LIN {X 0,Y 397.224,Z 668.821,A -85,B 0,C 180,E1 -11416.703,E2 -11416.703} C_VEL
LIN {X 0,Y 397.214,Z 668.819,A -85,B 0,C 180,E1 -11419.809,E2 -11419.809} C_VEL
LIN {X 0,Y 397.36,Z 668.8,A -85,B 0,C 180,E1 -11422.888,E2 -11422.888} C_VEL
LIN {X 0,Y 397.212,Z 669.008,A -85,B 0,C 180,E1 -11425.433,E2 -11425.433} C_VEL
LIN {X 0,Y 397.512,Z 669.23,A -85,B 0,C 180,E1 -11427.974,E2 -11427.974} C_VEL
LIN {X 0,Y 397.665,Z 669.27,A -85,B 0,C 180,E1 -11430,E2 -11430} C_VEL
LIN {X 0,Y 397.41,Z 669.17,A -85,B 0,C 180,E1 -11433.041,E2 -11433.041} C_VEL
LIN {X 0,Y 397.36,Z 668.8,A -85,B 0,C 180,E1 -11437.112,E2 -11437.112} C_VEL
LIN {X 0,Y 397.214,Z 668.819,A -85,B 0,C 180,E1 -11440.191,E2 -11440.191} C_VEL
LIN {X 0,Y 397.222,Z 668.821,A -85,B 0,C 180,E1 -11443.321,E2 -11443.321} C_VEL
LIN {X 0,Y 397.177,Z 668.825,A -85,B 0,C 180,E1 -11447.155,E2 -11447.155} C_VEL
LIN {X 0,Y 397.098,Z 668.833,A -85,B 0,C 180,E1 -11450.73,E2 -11450.73} C_VEL
LIN {X 0,Y 397.128,Z 668.833,A -85,B 0,C 180,E1 -11454.018,E2 -11454.018} C_VEL
LIN {X 0,Y 397.129,Z 668.83,A -85,B 0,C 180,E1 -11456.329,E2 -11456.329} C_VEL
LIN {X 0,Y 396.46,Z 668.913,A -85,B 0,C 180,E1 -11457.176,E2 -11457.176} C_VEL
LIN {X 0,Y 393.587,Z 669.271,A -85,B 0,C 180,E1 -11458.552,E2 -11458.552} C_VEL
LIN {X 0,Y 391.15,Z 669.576,A -85,B 0,C 180,E1 -11459.663,E2 -11459.663} C_VEL
LIN {X 0,Y 390.098,Z 669.707,A -85,B 0,C 180,E1 -11460.523,E2 -11460.523} C_VEL
LIN {X 0,Y 390.01,Z 669.714,A -85,B 0,C 180,E1 -11460.814,E2 -11460.814} C_VEL
LIN {X 0,Y 390.062,Z 669.71,A -85,B 0,C 180,E1 -11464.024,E2 -11464.024} C_VEL
LIN {X 0,Y 390.04,Z 669.713,A -85,B 0,C 180,E1 -11467.551,E2 -11467.551} C_VEL
LIN {X 0,Y 390.07,Z 669.71,A -85,B 0,C 180,E1 -11470.824,E2 -11470.824} C_VEL
LIN {X 0,Y 390.052,Z 669.711,A -85,B 0,C 180,E1 -11473.886,E2 -11473.886} C_VEL
LIN {X 0,Y 390.108,Z 669.706,A -85,B 0,C 180,E1 -11476.797,E2 -11476.797} C_VEL
LIN {X 0,Y 390.07,Z 669.71,A -85,B 0,C 180,E1 -11479.563,E2 -11479.563} C_VEL
LIN {X 0,Y 390.039,Z 669.686,A -85,B 0,C 180,E1 -11482.448,E2 -11482.448} C_VEL
LIN {X 0,Y 390.059,Z 669.698,A -85,B 0,C 180,E1 -11485.975,E2 -11485.975} C_VEL
LIN {X 0,Y 390.042,Z 669.68,A -85,B 0,C 180,E1 -11489.868,E2 -11489.868} C_VEL
LIN {X 0,Y 390.104,Z 669.682,A -85,B 0,C 180,E1 -11493.232,E2 -11493.232} C_VEL
LIN {X 0,Y 390.102,Z 669.699,A -85,B 0,C 180,E1 -11496.748,E2 -11496.748} C_VEL
LIN {X 0,Y 390.121,Z 669.704,A -85,B 0,C 180,E1 -11499.984,E2 -11499.984} C_VEL
LIN {X 0,Y 390.128,Z 669.69,A -85,B 0,C 180,E1 -11503.248,E2 -11503.248} C_VEL
LIN {X 0,Y 390.185,Z 669.677,A -85,B 0,C 180,E1 -11506.562,E2 -11506.562} C_VEL
LIN {X 0,Y 390.199,Z 669.684,A -85,B 0,C 180,E1 -11510.671,E2 -11510.671} C_VEL
LIN {X 0,Y 390.328,Z 669.669,A -85,B 0,C 180,E1 -11513.798,E2 -11513.798} C_VEL
LIN {X 0,Y 390.411,Z 669.649,A -85,B 0,C 180,E1 -11517.937,E2 -11517.937} C_VEL
LIN {X 0,Y 390.542,Z 669.648,A -85,B 0,C 180,E1 -11520,E2 -11520} C_VEL
LIN {X 0,Y 390.308,Z 669.665,A -85,B 0,C 180,E1 -11523.097,E2 -11523.097} C_VEL
LIN {X 0,Y 390.33,Z 669.673,A -85,B 0,C 180,E1 -11526.202,E2 -11526.202} C_VEL
LIN {X 0,Y 390.201,Z 669.685,A -85,B 0,C 180,E1 -11529.329,E2 -11529.329} C_VEL
LIN {X 0,Y 390.17,Z 669.682,A -85,B 0,C 180,E1 -11532.483,E2 -11532.483} C_VEL
LIN {X 0,Y 390.131,Z 669.698,A -85,B 0,C 180,E1 -11535.677,E2 -11535.677} C_VEL
LIN {X 0,Y 390.108,Z 669.695,A -85,B 0,C 180,E1 -11538.922,E2 -11538.922} C_VEL
LIN {X 0,Y 390.032,Z 669.699,A -85,B 0,C 180,E1 -11542.235,E2 -11542.235} C_VEL
LIN {X 0,Y 390.111,Z 669.696,A -85,B 0,C 180,E1 -11545.744,E2 -11545.744} C_VEL
LIN {X 0,Y 390.056,Z 669.66,A -85,B 0,C 180,E1 -11549.11,E2 -11549.11} C_VEL
LIN {X 0,Y 390.037,Z 669.712,A -85,B 0,C 180,E1 -11552.722,E2 -11552.722} C_VEL
LIN {X 0,Y 390.051,Z 669.68,A -85,B 0,C 180,E1 -11555.826,E2 -11555.826} C_VEL
LIN {X 0,Y 390.069,Z 669.707,A -85,B 0,C 180,E1 -11559.22,E2 -11559.22} C_VEL
LIN {X 0,Y 390.117,Z 669.688,A -85,B 0,C 180,E1 -11562.388,E2 -11562.388} C_VEL
LIN {X 0,Y 390.059,Z 669.69,A -85,B 0,C 180,E1 -11565.358,E2 -11565.358} C_VEL
LIN {X 0,Y 390.068,Z 669.864,A -85,B 0,C 180,E1 -11569.083,E2 -11569.083} C_VEL
LIN {X 0,Y 393.041,Z 680.441,A -85,B 0,C 180,E1 -11571.884,E2 -11571.884} C_VEL
LIN {X 0,Y 395.697,Z 690.609,A -85,B 0,C 180,E1 -11574.336,E2 -11574.336} C_VEL
LIN {X 0,Y 404.177,Z 707.9,A -85,B 0,C 180,E1 -11575.584,E2 -11575.584} C_VEL
LIN {X 0,Y 406.863,Z 714.125,A -85,B 0,C 180,E1 -11575.97,E2 -11575.97} C_VEL
LIN {X 0,Y 412.259,Z 737.158,A -85,B 0,C 180,E1 -11576.941,E2 -11576.941} C_VEL
LIN {X 0,Y 409.574,Z 850.002,A -85,B 0,C 180,E1 -11578.982,E2 -11578.982} C_VEL
LIN {X 0,Y 408.459,Z 894.918,A -85,B 0,C 180,E1 -11579.824,E2 -11579.824} C_VEL
LIN {X 0,Y 407.68,Z 907.428,A -85,B 0,C 180,E1 -11580.148,E2 -11580.148} C_VEL
LIN {X 0,Y 406.718,Z 919.552,A -85,B 0,C 180,E1 -11580.569,E2 -11580.569} C_VEL
LIN {X 0,Y 405.755,Z 931.929,A -85,B 0,C 180,E1 -11581.131,E2 -11581.131} C_VEL
LIN {X 0,Y 404.553,Z 943.316,A -85,B 0,C 180,E1 -11581.746,E2 -11581.746} C_VEL
LIN {X 0,Y 402.984,Z 957.059,A -85,B 0,C 180,E1 -11582.657,E2 -11582.657} C_VEL
LIN {X 0,Y 401.59,Z 968.362,A -85,B 0,C 180,E1 -11583.546,E2 -11583.546} C_VEL
LIN {X 0,Y 399.899,Z 980.294,A -85,B 0,C 180,E1 -11584.636,E2 -11584.636} C_VEL
LIN {X 0,Y 398.332,Z 991.097,A -85,B 0,C 180,E1 -11585.782,E2 -11585.782} C_VEL
LIN {X 0,Y 396.667,Z 1002.013,A -85,B 0,C 180,E1 -11587.119,E2 -11587.119} C_VEL
LIN {X 0,Y 395.292,Z 1010.87,A -85,B 0,C 180,E1 -11588.352,E2 -11588.352} C_VEL
LIN {X 0,Y 393.836,Z 1020.607,A -85,B 0,C 180,E1 -11589.909,E2 -11589.909} C_VEL
LIN {X 0,Y 392.506,Z 1029.848,A -85,B 0,C 180,E1 -11591.62,E2 -11591.62} C_VEL
LIN {X 0,Y 391.471,Z 1037.738,A -85,B 0,C 180,E1 -11593.307,E2 -11593.307} C_VEL
LIN {X 0,Y 390.576,Z 1044.167,A -85,B 0,C 180,E1 -11594.876,E2 -11594.876} C_VEL
LIN {X 0,Y 389.798,Z 1051.393,A -85,B 0,C 180,E1 -11596.964,E2 -11596.964} C_VEL
LIN {X 0,Y 389.384,Z 1056.079,A -85,B 0,C 180,E1 -11598.549,E2 -11598.549} C_VEL
LIN {X 0,Y 388.957,Z 1061.172,A -85,B 0,C 180,E1 -11600.641,E2 -11600.641} C_VEL
LIN {X 0,Y 388.806,Z 1065.168,A -85,B 0,C 180,E1 -11602.731,E2 -11602.731} C_VEL
LIN {X 0,Y 388.737,Z 1067.048,A -85,B 0,C 180,E1 -11603.905,E2 -11603.905} C_VEL
LIN {X 0,Y 388.657,Z 1069.301,A -85,B 0,C 180,E1 -11605.852,E2 -11605.852} C_VEL
LIN {X 0,Y 388.649,Z 1070.765,A -85,B 0,C 180,E1 -11607.927,E2 -11607.927} C_VEL
LIN {X 0,Y 388.704,Z 1071.251,A -85,B 0,C 180,E1 -11610,E2 -11610} C_VEL
LIN {X 0,Y 388.649,Z 1070.765,A -85,B 0,C 180,E1 -11612.073,E2 -11612.073} C_VEL
LIN {X 0,Y 388.657,Z 1069.301,A -85,B 0,C 180,E1 -11614.148,E2 -11614.148} C_VEL
LIN {X 0,Y 388.757,Z 1066.839,A -85,B 0,C 180,E1 -11616.227,E2 -11616.227} C_VEL
LIN {X 0,Y 388.897,Z 1062.26,A -85,B 0,C 180,E1 -11618.836,E2 -11618.836} C_VEL
LIN {X 0,Y 389.073,Z 1058.772,A -85,B 0,C 180,E1 -11620.406,E2 -11620.406} C_VEL
LIN {X 0,Y 389.66,Z 1053.051,A -85,B 0,C 180,E1 -11622.499,E2 -11622.499} C_VEL
LIN {X 0,Y 390.151,Z 1047.991,A -85,B 0,C 180,E1 -11624.074,E2 -11624.074} C_VEL
LIN {X 0,Y 391.109,Z 1039.958,A -85,B 0,C 180,E1 -11626.172,E2 -11626.172} C_VEL
LIN {X 0,Y 392.109,Z 1032.976,A -85,B 0,C 180,E1 -11627.74,E2 -11627.74} C_VEL
LIN {X 0,Y 393.19,Z 1025.004,A -85,B 0,C 180,E1 -11629.309,E2 -11629.309} C_VEL
LIN {X 0,Y 394.569,Z 1015.889,A -85,B 0,C 180,E1 -11630.869,E2 -11630.869} C_VEL
LIN {X 0,Y 396.135,Z 1005.854,A -85,B 0,C 180,E1 -11632.359,E2 -11632.359} C_VEL
LIN {X 0,Y 397.641,Z 995.45,A -85,B 0,C 180,E1 -11633.708,E2 -11633.708} C_VEL
LIN {X 0,Y 399.365,Z 984.036,A -85,B 0,C 180,E1 -11634.982,E2 -11634.982} C_VEL
LIN {X 0,Y 400.786,Z 973.609,A -85,B 0,C 180,E1 -11636,E2 -11636} C_VEL
LIN {X 0,Y 402.435,Z 961.583,A -85,B 0,C 180,E1 -11637.003,E2 -11637.003} C_VEL
LIN {X 0,Y 403.884,Z 949.459,A -85,B 0,C 180,E1 -11637.867,E2 -11637.867} C_VEL
LIN {X 0,Y 405.278,Z 936.716,A -85,B 0,C 180,E1 -11638.623,E2 -11638.623} C_VEL
LIN {X 0,Y 406.417,Z 923.283,A -85,B 0,C 180,E1 -11639.278,E2 -11639.278} C_VEL
LIN {X 0,Y 407.461,Z 910.365,A -85,B 0,C 180,E1 -11639.763,E2 -11639.763} C_VEL
LIN {X 0,Y 408.373,Z 896.659,A -85,B 0,C 180,E1 -11640.139,E2 -11640.139} C_VEL
LIN {X 0,Y 409.085,Z 870.937,A -85,B 0,C 180,E1 -11640.64,E2 -11640.64} C_VEL
LIN {X 0,Y 412.265,Z 737.158,A -85,B 0,C 180,E1 -11643.059,E2 -11643.059} C_VEL
LIN {X 0,Y 406.66,Z 713.318,A -85,B 0,C 180,E1 -11644.065,E2 -11644.065} C_VEL
LIN {X 0,Y 397.258,Z 693.815,A -85,B 0,C 180,E1 -11645.402,E2 -11645.402} C_VEL
LIN {X 0,Y 395.726,Z 690.524,A -85,B 0,C 180,E1 -11645.67,E2 -11645.67} C_VEL
LIN {X 0,Y 391.984,Z 676.49,A -85,B 0,C 180,E1 -11649.122,E2 -11649.122} C_VEL
LIN {X 0,Y 390.049,Z 669.745,A -85,B 0,C 180,E1 -11650.968,E2 -11650.968} C_VEL
LIN {X 0,Y 390.059,Z 669.689,A -85,B 0,C 180,E1 -11654.642,E2 -11654.642} C_VEL
LIN {X 0,Y 390.117,Z 669.688,A -85,B 0,C 180,E1 -11657.612,E2 -11657.612} C_VEL
LIN {X 0,Y 390.09,Z 669.705,A -85,B 0,C 180,E1 -11660.908,E2 -11660.908} C_VEL
LIN {X 0,Y 390.079,Z 669.679,A -85,B 0,C 180,E1 -11664.792,E2 -11664.792} C_VEL
LIN {X 0,Y 390.02,Z 669.706,A -85,B 0,C 180,E1 -11668.495,E2 -11668.495} C_VEL
LIN {X 0,Y 390.11,Z 669.657,A -85,B 0,C 180,E1 -11672.069,E2 -11672.069} C_VEL
LIN {X 0,Y 390.072,Z 669.707,A -85,B 0,C 180,E1 -11675.519,E2 -11675.519} C_VEL
LIN {X 0,Y 390.057,Z 669.708,A -85,B 0,C 180,E1 -11678.878,E2 -11678.878} C_VEL
LIN {X 0,Y 390.122,Z 669.689,A -85,B 0,C 180,E1 -11682.166,E2 -11682.166} C_VEL
LIN {X 0,Y 390.138,Z 669.695,A -85,B 0,C 180,E1 -11685.392,E2 -11685.392} C_VEL
LIN {X 0,Y 390.152,Z 669.692,A -85,B 0,C 180,E1 -11688.571,E2 -11688.571} C_VEL
LIN {X 0,Y 390.299,Z 669.66,A -85,B 0,C 180,E1 -11692.03,E2 -11692.03} C_VEL
LIN {X 0,Y 390.225,Z 669.688,A -85,B 0,C 180,E1 -11694.833,E2 -11694.833} C_VEL
LIN {X 0,Y 390.411,Z 669.654,A -85,B 0,C 180,E1 -11697.936,E2 -11697.936} C_VEL
LIN {X 0,Y 390.542,Z 669.647,A -85,B 0,C 180,E1 -11700,E2 -11700} C_VEL
LIN {X 0,Y 390.308,Z 669.662,A -85,B 0,C 180,E1 -11703.096,E2 -11703.096} C_VEL
LIN {X 0,Y 390.3,Z 669.67,A -85,B 0,C 180,E1 -11706.58,E2 -11706.58} C_VEL
LIN {X 0,Y 390.199,Z 669.686,A -85,B 0,C 180,E1 -11709.329,E2 -11709.329} C_VEL
LIN {X 0,Y 390.185,Z 669.678,A -85,B 0,C 180,E1 -11713.438,E2 -11713.438} C_VEL
LIN {X 0,Y 390.139,Z 669.687,A -85,B 0,C 180,E1 -11717.308,E2 -11717.308} C_VEL
LIN {X 0,Y 390.106,Z 669.702,A -85,B 0,C 180,E1 -11720.481,E2 -11720.481} C_VEL
LIN {X 0,Y 390.101,Z 669.699,A -85,B 0,C 180,E1 -11723.35,E2 -11723.35} C_VEL
LIN {X 0,Y 390.104,Z 669.681,A -85,B 0,C 180,E1 -11726.768,E2 -11726.768} C_VEL
LIN {X 0,Y 390.034,Z 669.684,A -85,B 0,C 180,E1 -11730.3,E2 -11730.3} C_VEL
LIN {X 0,Y 390.059,Z 669.698,A -85,B 0,C 180,E1 -11734.025,E2 -11734.025} C_VEL
LIN {X 0,Y 390.039,Z 669.686,A -85,B 0,C 180,E1 -11737.552,E2 -11737.552} C_VEL
LIN {X 0,Y 390.075,Z 669.71,A -85,B 0,C 180,E1 -11740.826,E2 -11740.826} C_VEL
LIN {X 0,Y 390.096,Z 669.706,A -85,B 0,C 180,E1 -11743.894,E2 -11743.894} C_VEL
LIN {X 0,Y 390.073,Z 669.71,A -85,B 0,C 180,E1 -11747.62,E2 -11747.62} C_VEL
LIN {X 0,Y 390.088,Z 669.708,A -85,B 0,C 180,E1 -11750.909,E2 -11750.909} C_VEL
LIN {X 0,Y 390.079,Z 669.708,A -85,B 0,C 180,E1 -11754.794,E2 -11754.794} C_VEL
LIN {X 0,Y 390.021,Z 669.714,A -85,B 0,C 180,E1 -11758.496,E2 -11758.496} C_VEL
LIN {X 0,Y 390.112,Z 669.705,A -85,B 0,C 180,E1 -11762.07,E2 -11762.07} C_VEL
LIN {X 0,Y 390.075,Z 669.708,A -85,B 0,C 180,E1 -11765.52,E2 -11765.52} C_VEL
LIN {X 0,Y 390.051,Z 669.712,A -85,B 0,C 180,E1 -11768.878,E2 -11768.878} C_VEL
LIN {X 0,Y 390.124,Z 669.702,A -85,B 0,C 180,E1 -11772.167,E2 -11772.167} C_VEL
LIN {X 0,Y 390.14,Z 669.731,A -85,B 0,C 180,E1 -11775.393,E2 -11775.393} C_VEL
LIN {X 0,Y 390.278,Z 670.28,A -85,B 0,C 180,E1 -11776.757,E2 -11776.757} C_VEL
LIN {X 0,Y 390.794,Z 671.827,A -85,B 0,C 180,E1 -11777.867,E2 -11777.867} C_VEL
LIN {X 0,Y 392.016,Z 673.68,A -85,B 0,C 180,E1 -11779.411,E2 -11779.411} C_VEL
LIN {X 0,Y 393.321,Z 674.699,A -85,B 0,C 180,E1 -11781.264,E2 -11781.264} C_VEL
LIN {X 0,Y 394.824,Z 675.448,A -85,B 0,C 180,E1 -11783.869,E2 -11783.869} C_VEL
LIN {X 0,Y 395.643,Z 676.056,A -85,B 0,C 180,E1 -11785.926,E2 -11785.926} C_VEL
LIN {X 0,Y 396.111,Z 676.191,A -85,B 0,C 180,E1 -11787.966,E2 -11787.966} C_VEL
LIN {X 0,Y 396.315,Z 676.238,A -85,B 0,C 180,E1 -11790,E2 -11790} C_VEL
LIN {X 0,Y 396.112,Z 676.191,A -85,B 0,C 180,E1 -11792.034,E2 -11792.034} C_VEL
LIN {X 0,Y 395.45,Z 675.884,A -85,B 0,C 180,E1 -11794.587,E2 -11794.587} C_VEL
LIN {X 0,Y 394.284,Z 675.199,A -85,B 0,C 180,E1 -11797.167,E2 -11797.167} C_VEL
LIN {X 0,Y 392.652,Z 674.256,A -85,B 0,C 180,E1 -11799.699,E2 -11799.699} C_VEL
LIN {X 0,Y 391.359,Z 672.872,A -85,B 0,C 180,E1 -11801.393,E2 -11801.393} C_VEL
LIN {X 0,Y 390.326,Z 670.548,A -85,B 0,C 180,E1 -11802.973,E2 -11802.973} C_VEL
LIN {X 0,Y 390.138,Z 669.78,A -85,B 0,C 180,E1 -11804.075,E2 -11804.075} C_VEL
LIN {X 0,Y 390.144,Z 669.702,A -85,B 0,C 180,E1 -11807.307,E2 -11807.307} C_VEL
LIN {X 0,Y 390.082,Z 669.707,A -85,B 0,C 180,E1 -11810.47,E2 -11810.47} C_VEL
LIN {X 0,Y 390.084,Z 669.707,A -85,B 0,C 180,E1 -11813.35,E2 -11813.35} C_VEL
LIN {X 0,Y 390.108,Z 669.706,A -85,B 0,C 180,E1 -11816.768,E2 -11816.768} C_VEL
LIN {X 0,Y 390.038,Z 669.713,A -85,B 0,C 180,E1 -11820.299,E2 -11820.299} C_VEL
LIN {X 0,Y 390.01,Z 669.714,A -85,B 0,C 180,E1 -11820.814,E2 -11820.814} C_VEL
LIN {X 0,Y 389.336,Z 669.8,A -85,B 0,C 180,E1 -11821.676,E2 -11821.676} C_VEL
LIN {X 0,Y 386.486,Z 670.155,A -85,B 0,C 180,E1 -11823.078,E2 -11823.078} C_VEL
LIN {X 0,Y 384.087,Z 670.454,A -85,B 0,C 180,E1 -11824.211,E2 -11824.211} C_VEL
LIN {X 0,Y 383.069,Z 670.582,A -85,B 0,C 180,E1 -11825.087,E2 -11825.087} C_VEL
LIN {X 0,Y 382.993,Z 670.588,A -85,B 0,C 180,E1 -11825.383,E2 -11825.383} C_VEL
LIN {X 0,Y 383.001,Z 670.59,A -85,B 0,C 180,E1 -11828.6,E2 -11828.6} C_VEL
LIN {X 0,Y 383.006,Z 670.589,A -85,B 0,C 180,E1 -11831.343,E2 -11831.343} C_VEL
LIN {X 0,Y 383,Z 670.591,A -85,B 0,C 180,E1 -11834.305,E2 -11834.305} C_VEL
LIN {X 0,Y 383.067,Z 670.583,A -85,B 0,C 180,E1 -11837.249,E2 -11837.249} C_VEL
LIN {X 0,Y 383.014,Z 670.588,A -85,B 0,C 180,E1 -11840.412,E2 -11840.412} C_VEL
LIN {X 0,Y 383.018,Z 670.546,A -85,B 0,C 180,E1 -11844.044,E2 -11844.044} C_VEL
LIN {X 0,Y 382.979,Z 670.593,A -85,B 0,C 180,E1 -11847.577,E2 -11847.577} C_VEL
LIN {X 0,Y 382.987,Z 670.549,A -85,B 0,C 180,E1 -11850.3,E2 -11850.3} C_VEL
LIN {X 0,Y 383.047,Z 670.548,A -85,B 0,C 180,E1 -11852.698,E2 -11852.698} C_VEL
LIN {X 0,Y 383.034,Z 670.581,A -85,B 0,C 180,E1 -11856.193,E2 -11856.193} C_VEL
LIN {X 0,Y 383.072,Z 670.579,A -85,B 0,C 180,E1 -11859.6,E2 -11859.6} C_VEL
LIN {X 0,Y 383.095,Z 670.565,A -85,B 0,C 180,E1 -11862.931,E2 -11862.931} C_VEL
LIN {X 0,Y 383.116,Z 670.558,A -85,B 0,C 180,E1 -11866.464,E2 -11866.464} C_VEL
LIN {X 0,Y 383.145,Z 670.565,A -85,B 0,C 180,E1 -11870.498,E2 -11870.498} C_VEL
LIN {X 0,Y 383.282,Z 670.546,A -85,B 0,C 180,E1 -11873.684,E2 -11873.684} C_VEL
LIN {X 0,Y 383.379,Z 670.524,A -85,B 0,C 180,E1 -11877.899,E2 -11877.899} C_VEL
LIN {X 0,Y 383.511,Z 670.524,A -85,B 0,C 180,E1 -11880,E2 -11880} C_VEL
LIN {X 0,Y 383.244,Z 670.544,A -85,B 0,C 180,E1 -11883.154,E2 -11883.154} C_VEL
LIN {X 0,Y 383.284,Z 670.551,A -85,B 0,C 180,E1 -11886.317,E2 -11886.317} C_VEL
LIN {X 0,Y 383.148,Z 670.566,A -85,B 0,C 180,E1 -11889.502,E2 -11889.502} C_VEL
LIN {X 0,Y 383.133,Z 670.557,A -85,B 0,C 180,E1 -11892.716,E2 -11892.716} C_VEL
LIN {X 0,Y 383.072,Z 670.576,A -85,B 0,C 180,E1 -11895.974,E2 -11895.974} C_VEL
LIN {X 0,Y 383.063,Z 670.576,A -85,B 0,C 180,E1 -11899.284,E2 -11899.284} C_VEL
LIN {X 0,Y 383,Z 670.574,A -85,B 0,C 180,E1 -11902.665,E2 -11902.665} C_VEL
LIN {X 0,Y 383.072,Z 670.569,A -85,B 0,C 180,E1 -11906.124,E2 -11906.124} C_VEL
LIN {X 0,Y 383.042,Z 670.532,A -85,B 0,C 180,E1 -11908.493,E2 -11908.493} C_VEL
LIN {X 0,Y 383.004,Z 670.589,A -85,B 0,C 180,E1 -11912.15,E2 -11912.15} C_VEL
LIN {X 0,Y 383.011,Z 670.565,A -85,B 0,C 180,E1 -11914.669,E2 -11914.669} C_VEL
LIN {X 0,Y 382.998,Z 670.585,A -85,B 0,C 180,E1 -11917.905,E2 -11917.905} C_VEL
LIN {X 0,Y 383.041,Z 670.558,A -85,B 0,C 180,E1 -11921.34,E2 -11921.34} C_VEL
LIN {X 0,Y 383.032,Z 670.575,A -85,B 0,C 180,E1 -11924.31,E2 -11924.31} C_VEL
LIN {X 0,Y 382.983,Z 670.585,A -85,B 0,C 180,E1 -11927.95,E2 -11927.95} C_VEL
LIN {X 0,Y 383.025,Z 670.88,A -85,B 0,C 180,E1 -11928.499,E2 -11928.499} C_VEL
LIN {X 0,Y 386.182,Z 681.98,A -85,B 0,C 180,E1 -11931.494,E2 -11931.494} C_VEL
LIN {X 0,Y 388.446,Z 690.413,A -85,B 0,C 180,E1 -11933.574,E2 -11933.574} C_VEL
LIN {X 0,Y 397.258,Z 708.158,A -85,B 0,C 180,E1 -11934.908,E2 -11934.908} C_VEL
LIN {X 0,Y 401.315,Z 717.115,A -85,B 0,C 180,E1 -11935.502,E2 -11935.502} C_VEL
LIN {X 0,Y 406.335,Z 738.734,A -85,B 0,C 180,E1 -11936.432,E2 -11936.432} C_VEL
LIN {X 0,Y 402.43,Z 891.118,A -85,B 0,C 180,E1 -11939.23,E2 -11939.23} C_VEL
LIN {X 0,Y 401.727,Z 904.285,A -85,B 0,C 180,E1 -11939.55,E2 -11939.55} C_VEL
LIN {X 0,Y 400.613,Z 918.6,A -85,B 0,C 180,E1 -11940.039,E2 -11940.039} C_VEL
LIN {X 0,Y 399.502,Z 931.722,A -85,B 0,C 180,E1 -11940.636,E2 -11940.636} C_VEL
LIN {X 0,Y 398.284,Z 943.109,A -85,B 0,C 180,E1 -11941.26,E2 -11941.26} C_VEL
LIN {X 0,Y 396.71,Z 956.348,A -85,B 0,C 180,E1 -11942.145,E2 -11942.145} C_VEL
LIN {X 0,Y 395.136,Z 968.521,A -85,B 0,C 180,E1 -11943.116,E2 -11943.116} C_VEL
LIN {X 0,Y 393.43,Z 980.087,A -85,B 0,C 180,E1 -11944.189,E2 -11944.189} C_VEL
LIN {X 0,Y 391.774,Z 990.889,A -85,B 0,C 180,E1 -11945.35,E2 -11945.35} C_VEL
LIN {X 0,Y 390.124,Z 1001.391,A -85,B 0,C 180,E1 -11946.652,E2 -11946.652} C_VEL
LIN {X 0,Y 388.608,Z 1010.662,A -85,B 0,C 180,E1 -11947.96,E2 -11947.96} C_VEL
LIN {X 0,Y 387.069,Z 1020.398,A -85,B 0,C 180,E1 -11949.543,E2 -11949.543} C_VEL
LIN {X 0,Y 385.72,Z 1029.432,A -85,B 0,C 180,E1 -11951.24,E2 -11951.24} C_VEL
LIN {X 0,Y 384.597,Z 1037.53,A -85,B 0,C 180,E1 -11953,E2 -11953} C_VEL
LIN {X 0,Y 383.627,Z 1043.959,A -85,B 0,C 180,E1 -11954.596,E2 -11954.596} C_VEL
LIN {X 0,Y 382.827,Z 1050.972,A -85,B 0,C 180,E1 -11956.651,E2 -11956.651} C_VEL
LIN {X 0,Y 382.343,Z 1055.871,A -85,B 0,C 180,E1 -11958.335,E2 -11958.335} C_VEL
LIN {X 0,Y 381.898,Z 1060.965,A -85,B 0,C 180,E1 -11960.467,E2 -11960.467} C_VEL
LIN {X 0,Y 381.708,Z 1064.961,A -85,B 0,C 180,E1 -11962.595,E2 -11962.595} C_VEL
LIN {X 0,Y 381.655,Z 1067.021,A -85,B 0,C 180,E1 -11963.924,E2 -11963.924} C_VEL
LIN {X 0,Y 381.582,Z 1069.095,A -85,B 0,C 180,E1 -11965.775,E2 -11965.775} C_VEL
LIN {X 0,Y 381.547,Z 1070.559,A -85,B 0,C 180,E1 -11967.889,E2 -11967.889} C_VEL
LIN {X 0,Y 381.635,Z 1071.047,A -85,B 0,C 180,E1 -11970,E2 -11970} C_VEL
LIN {X 0,Y 381.547,Z 1070.559,A -85,B 0,C 180,E1 -11972.111,E2 -11972.111} C_VEL
LIN {X 0,Y 381.582,Z 1069.095,A -85,B 0,C 180,E1 -11974.225,E2 -11974.225} C_VEL
LIN {X 0,Y 381.662,Z 1066.633,A -85,B 0,C 180,E1 -11976.343,E2 -11976.343} C_VEL
LIN {X 0,Y 381.821,Z 1062.052,A -85,B 0,C 180,E1 -11979.001,E2 -11979.001} C_VEL
LIN {X 0,Y 382.032,Z 1058.565,A -85,B 0,C 180,E1 -11980.6,E2 -11980.6} C_VEL
LIN {X 0,Y 382.65,Z 1052.843,A -85,B 0,C 180,E1 -11982.732,E2 -11982.732} C_VEL
LIN {X 0,Y 383.169,Z 1047.782,A -85,B 0,C 180,E1 -11984.336,E2 -11984.336} C_VEL
LIN {X 0,Y 384.207,Z 1039.75,A -85,B 0,C 180,E1 -11986.47,E2 -11986.47} C_VEL
LIN {X 0,Y 385.206,Z 1032.766,A -85,B 0,C 180,E1 -11988.068,E2 -11988.068} C_VEL
LIN {X 0,Y 386.381,Z 1024.795,A -85,B 0,C 180,E1 -11989.663,E2 -11989.663} C_VEL
LIN {X 0,Y 387.837,Z 1015.681,A -85,B 0,C 180,E1 -11991.248,E2 -11991.248} C_VEL
LIN {X 0,Y 389.42,Z 1006.053,A -85,B 0,C 180,E1 -11992.706,E2 -11992.706} C_VEL
LIN {X 0,Y 391.093,Z 995.242,A -85,B 0,C 180,E1 -11994.13,E2 -11994.13} C_VEL
LIN {X 0,Y 392.682,Z 985.075,A -85,B 0,C 180,E1 -11995.296,E2 -11995.296} C_VEL
LIN {X 0,Y 394.373,Z 973.402,A -85,B 0,C 180,E1 -11996.456,E2 -11996.456} C_VEL
LIN {X 0,Y 396.067,Z 961.376,A -85,B 0,C 180,E1 -11997.474,E2 -11997.474} C_VEL
LIN {X 0,Y 397.579,Z 949.053,A -85,B 0,C 180,E1 -11998.363,E2 -11998.363} C_VEL
LIN {X 0,Y 399.022,Z 936.509,A -85,B 0,C 180,E1 -11999.114,E2 -11999.114} C_VEL
LIN {X 0,Y 400.223,Z 923.077,A -85,B 0,C 180,E1 -11999.776,E2 -11999.776} C_VEL
LIN {X 0,Y 401.321,Z 910.16,A -85,B 0,C 180,E1 -12000.266,E2 -12000.266} C_VEL
LIN {X 0,Y 402.237,Z 896.826,A -85,B 0,C 180,E1 -12000.638,E2 -12000.638} C_VEL
LIN {X 0,Y 402.977,Z 871.625,A -85,B 0,C 180,E1 -12001.138,E2 -12001.138} C_VEL
LIN {X 0,Y 406.361,Z 738.759,A -85,B 0,C 180,E1 -12003.565,E2 -12003.565} C_VEL
LIN {X 0,Y 401.03,Z 716.167,A -85,B 0,C 180,E1 -12004.546,E2 -12004.546} C_VEL
LIN {X 0,Y 392.191,Z 697.813,A -85,B 0,C 180,E1 -12005.837,E2 -12005.837} C_VEL
LIN {X 0,Y 388.368,Z 690.209,A -85,B 0,C 180,E1 -12006.456,E2 -12006.456} C_VEL
LIN {X 0,Y 385.491,Z 679.253,A -85,B 0,C 180,E1 -12009.211,E2 -12009.211} C_VEL
LIN {X 0,Y 383.019,Z 670.855,A -85,B 0,C 180,E1 -12011.5,E2 -12011.5} C_VEL
LIN {X 0,Y 382.983,Z 670.585,A -85,B 0,C 180,E1 -12012.05,E2 -12012.05} C_VEL
LIN {X 0,Y 383.036,Z 670.576,A -85,B 0,C 180,E1 -12015.795,E2 -12015.795} C_VEL
LIN {X 0,Y 383.039,Z 670.558,A -85,B 0,C 180,E1 -12018.785,E2 -12018.785} C_VEL
LIN {X 0,Y 382.998,Z 670.585,A -85,B 0,C 180,E1 -12022.095,E2 -12022.095} C_VEL
LIN {X 0,Y 383.011,Z 670.565,A -85,B 0,C 180,E1 -12025.331,E2 -12025.331} C_VEL
LIN {X 0,Y 382.979,Z 670.572,A -85,B 0,C 180,E1 -12029.081,E2 -12029.081} C_VEL
LIN {X 0,Y 383.049,Z 670.546,A -85,B 0,C 180,E1 -12032.697,E2 -12032.697} C_VEL
LIN {X 0,Y 383.044,Z 670.583,A -85,B 0,C 180,E1 -12035.039,E2 -12035.039} C_VEL
LIN {X 0,Y 382.99,Z 670.581,A -85,B 0,C 180,E1 -12038.469,E2 -12038.469} C_VEL
LIN {X 0,Y 383.085,Z 670.565,A -85,B 0,C 180,E1 -12041.827,E2 -12041.827} C_VEL
LIN {X 0,Y 383.103,Z 670.574,A -85,B 0,C 180,E1 -12045.118,E2 -12045.118} C_VEL
LIN {X 0,Y 383.1,Z 670.568,A -85,B 0,C 180,E1 -12048.358,E2 -12048.358} C_VEL
LIN {X 0,Y 383.256,Z 670.537,A -85,B 0,C 180,E1 -12051.974,E2 -12051.974} C_VEL
LIN {X 0,Y 383.197,Z 670.563,A -85,B 0,C 180,E1 -12054.738,E2 -12054.738} C_VEL
LIN {X 0,Y 383.378,Z 670.529,A -85,B 0,C 180,E1 -12057.899,E2 -12057.899} C_VEL
LIN {X 0,Y 383.511,Z 670.523,A -85,B 0,C 180,E1 -12060,E2 -12060} C_VEL
LIN {X 0,Y 383.245,Z 670.542,A -85,B 0,C 180,E1 -12063.153,E2 -12063.153} C_VEL
LIN {X 0,Y 383.261,Z 670.547,A -85,B 0,C 180,E1 -12066.569,E2 -12066.569} C_VEL
LIN {X 0,Y 383.145,Z 670.566,A -85,B 0,C 180,E1 -12069.502,E2 -12069.502} C_VEL
LIN {X 0,Y 383.116,Z 670.559,A -85,B 0,C 180,E1 -12073.536,E2 -12073.536} C_VEL
LIN {X 0,Y 383.086,Z 670.564,A -85,B 0,C 180,E1 -12077.455,E2 -12077.455} C_VEL
LIN {X 0,Y 383.053,Z 670.579,A -85,B 0,C 180,E1 -12080.66,E2 -12080.66} C_VEL
LIN {X 0,Y 383.034,Z 670.581,A -85,B 0,C 180,E1 -12083.807,E2 -12083.807} C_VEL
LIN {X 0,Y 383.047,Z 670.548,A -85,B 0,C 180,E1 -12087.302,E2 -12087.302} C_VEL
LIN {X 0,Y 382.977,Z 670.573,A -85,B 0,C 180,E1 -12090.918,E2 -12090.918} C_VEL
LIN {X 0,Y 383.009,Z 670.562,A -85,B 0,C 180,E1 -12094.668,E2 -12094.668} C_VEL
LIN {X 0,Y 382.995,Z 670.57,A -85,B 0,C 180,E1 -12097.905,E2 -12097.905} C_VEL
LIN {X 0,Y 383.039,Z 670.586,A -85,B 0,C 180,E1 -12101.339,E2 -12101.339} C_VEL
LIN {X 0,Y 383.027,Z 670.586,A -85,B 0,C 180,E1 -12104.31,E2 -12104.31} C_VEL
LIN {X 0,Y 383.032,Z 670.586,A -85,B 0,C 180,E1 -12107.245,E2 -12107.245} C_VEL
LIN {X 0,Y 383.014,Z 670.587,A -85,B 0,C 180,E1 -12110.413,E2 -12110.413} C_VEL
LIN {X 0,Y 383.02,Z 670.587,A -85,B 0,C 180,E1 -12114.045,E2 -12114.045} C_VEL
LIN {X 0,Y 382.982,Z 670.593,A -85,B 0,C 180,E1 -12117.578,E2 -12117.578} C_VEL
LIN {X 0,Y 382.992,Z 670.592,A -85,B 0,C 180,E1 -12120.301,E2 -12120.301} C_VEL
LIN {X 0,Y 383.051,Z 670.583,A -85,B 0,C 180,E1 -12122.699,E2 -12122.699} C_VEL
LIN {X 0,Y 383.047,Z 670.584,A -85,B 0,C 180,E1 -12125.04,E2 -12125.04} C_VEL
LIN {X 0,Y 382.988,Z 670.592,A -85,B 0,C 180,E1 -12128.469,E2 -12128.469} C_VEL
LIN {X 0,Y 383.088,Z 670.839,A -85,B 0,C 180,E1 -12130.996,E2 -12130.996} C_VEL
LIN {X 0,Y 383.519,Z 672.313,A -85,B 0,C 180,E1 -12131.957,E2 -12131.957} C_VEL
LIN {X 0,Y 384.908,Z 674.478,A -85,B 0,C 180,E1 -12133.151,E2 -12133.151} C_VEL
LIN {X 0,Y 386.874,Z 676.015,A -85,B 0,C 180,E1 -12134.822,E2 -12134.822} C_VEL
LIN {X 0,Y 388.937,Z 677.277,A -85,B 0,C 180,E1 -12136.711,E2 -12136.711} C_VEL
LIN {X 0,Y 390.561,Z 680.095,A -85,B 0,C 180,E1 -12138.715,E2 -12138.715} C_VEL
LIN {X 0,Y 392.104,Z 681.548,A -85,B 0,C 180,E1 -12140.717,E2 -12140.717} C_VEL
LIN {X 0,Y 393.72,Z 682.4,A -85,B 0,C 180,E1 -12143.337,E2 -12143.337} C_VEL
LIN {X 0,Y 394.776,Z 683.078,A -85,B 0,C 180,E1 -12145.917,E2 -12145.917} C_VEL
LIN {X 0,Y 395.246,Z 683.238,A -85,B 0,C 180,E1 -12147.962,E2 -12147.962} C_VEL
LIN {X 0,Y 395.45,Z 683.285,A -85,B 0,C 180,E1 -12150,E2 -12150} C_VEL
LIN {X 0,Y 395.246,Z 683.239,A -85,B 0,C 180,E1 -12152.038,E2 -12152.038} C_VEL
LIN {X 0,Y 394.58,Z 682.93,A -85,B 0,C 180,E1 -12154.597,E2 -12154.597} C_VEL
LIN {X 0,Y 393.407,Z 682.244,A -85,B 0,C 180,E1 -12157.184,E2 -12157.184} C_VEL
LIN {X 0,Y 391.762,Z 681.307,A -85,B 0,C 180,E1 -12159.721,E2 -12159.721} C_VEL
LIN {X 0,Y 390.357,Z 679.813,A -85,B 0,C 180,E1 -12161.554,E2 -12161.554} C_VEL
LIN {X 0,Y 388.611,Z 676.952,A -85,B 0,C 180,E1 -12163.597,E2 -12163.597} C_VEL
LIN {X 0,Y 385.769,Z 675.309,A -85,B 0,C 180,E1 -12166.13,E2 -12166.13} C_VEL
LIN {X 0,Y 384.08,Z 673.407,A -85,B 0,C 180,E1 -12167.545,E2 -12167.545} C_VEL
LIN {X 0,Y 383.189,Z 671.308,A -85,B 0,C 180,E1 -12168.582,E2 -12168.582} C_VEL
LIN {X 0,Y 383.056,Z 670.66,A -85,B 0,C 180,E1 -12169.283,E2 -12169.283} C_VEL
LIN {X 0,Y 383.004,Z 670.592,A -85,B 0,C 180,E1 -12172.664,E2 -12172.664} C_VEL
LIN {X 0,Y 383.075,Z 670.58,A -85,B 0,C 180,E1 -12176.123,E2 -12176.123} C_VEL
LIN {X 0,Y 383.044,Z 670.584,A -85,B 0,C 180,E1 -12178.492,E2 -12178.492} C_VEL
LIN {X 0,Y 383.005,Z 670.591,A -85,B 0,C 180,E1 -12182.149,E2 -12182.149} C_VEL
LIN {X 0,Y 382.993,Z 670.588,A -85,B 0,C 180,E1 -12185.383,E2 -12185.383} C_VEL
LIN {X 0,Y 382.352,Z 670.672,A -85,B 0,C 180,E1 -12186.261,E2 -12186.261} C_VEL
LIN {X 0,Y 379.544,Z 671.022,A -85,B 0,C 180,E1 -12187.689,E2 -12187.689} C_VEL
LIN {X 0,Y 377.139,Z 671.321,A -85,B 0,C 180,E1 -12188.843,E2 -12188.843} C_VEL
LIN {X 0,Y 376.084,Z 671.451,A -85,B 0,C 180,E1 -12189.735,E2 -12189.735} C_VEL
LIN {X 0,Y 375.986,Z 671.462,A -85,B 0,C 180,E1 -12190.038,E2 -12190.038} C_VEL
LIN {X 0,Y 375.938,Z 671.469,A -85,B 0,C 180,E1 -12193.763,E2 -12193.763} C_VEL
LIN {X 0,Y 375.981,Z 671.466,A -85,B 0,C 180,E1 -12196.801,E2 -12196.801} C_VEL
LIN {X 0,Y 375.991,Z 671.462,A -85,B 0,C 180,E1 -12200.027,E2 -12200.027} C_VEL
LIN {X 0,Y 375.957,Z 671.424,A -85,B 0,C 180,E1 -12203.495,E2 -12203.495} C_VEL
LIN {X 0,Y 375.951,Z 671.451,A -85,B 0,C 180,E1 -12205.888,E2 -12205.888} C_VEL
LIN {X 0,Y 375.959,Z 671.434,A -85,B 0,C 180,E1 -12209.687,E2 -12209.687} C_VEL
LIN {X 0,Y 375.993,Z 671.416,A -85,B 0,C 180,E1 -12212.142,E2 -12212.142} C_VEL
LIN {X 0,Y 375.998,Z 671.458,A -85,B 0,C 180,E1 -12214.539,E2 -12214.539} C_VEL
LIN {X 0,Y 375.985,Z 671.452,A -85,B 0,C 180,E1 -12218.048,E2 -12218.048} C_VEL
LIN {X 0,Y 376.022,Z 671.449,A -85,B 0,C 180,E1 -12221.474,E2 -12221.474} C_VEL
LIN {X 0,Y 376.048,Z 671.452,A -85,B 0,C 180,E1 -12224.833,E2 -12224.833} C_VEL
LIN {X 0,Y 376.041,Z 671.442,A -85,B 0,C 180,E1 -12228.137,E2 -12228.137} C_VEL
LIN {X 0,Y 376.209,Z 671.419,A -85,B 0,C 180,E1 -12231.919,E2 -12231.919} C_VEL
LIN {X 0,Y 376.168,Z 671.441,A -85,B 0,C 180,E1 -12234.64,E2 -12234.64} C_VEL
LIN {X 0,Y 376.345,Z 671.4,A -85,B 0,C 180,E1 -12237.86,E2 -12237.86} C_VEL
LIN {X 0,Y 376.481,Z 671.4,A -85,B 0,C 180,E1 -12240,E2 -12240} C_VEL
LIN {X 0,Y 376.182,Z 671.424,A -85,B 0,C 180,E1 -12243.213,E2 -12243.213} C_VEL
LIN {X 0,Y 376.241,Z 671.426,A -85,B 0,C 180,E1 -12246.435,E2 -12246.435} C_VEL
LIN {X 0,Y 376.116,Z 671.443,A -85,B 0,C 180,E1 -12249.682,E2 -12249.682} C_VEL
LIN {X 0,Y 376.081,Z 671.438,A -85,B 0,C 180,E1 -12253.658,E2 -12253.658} C_VEL
LIN {X 0,Y 376.036,Z 671.442,A -85,B 0,C 180,E1 -12257.608,E2 -12257.608} C_VEL
LIN {X 0,Y 375.999,Z 671.461,A -85,B 0,C 180,E1 -12260.844,E2 -12260.844} C_VEL
LIN {X 0,Y 375.986,Z 671.463,A -85,B 0,C 180,E1 -12264.282,E2 -12264.282} C_VEL
LIN {X 0,Y 376.012,Z 671.438,A -85,B 0,C 180,E1 -12266.653,E2 -12266.653} C_VEL
LIN {X 0,Y 375.969,Z 671.411,A -85,B 0,C 180,E1 -12269.079,E2 -12269.079} C_VEL
LIN {X 0,Y 375.943,Z 671.468,A -85,B 0,C 180,E1 -12272.829,E2 -12272.829} C_VEL
LIN {X 0,Y 375.952,Z 671.435,A -85,B 0,C 180,E1 -12275.416,E2 -12275.416} C_VEL
LIN {X 0,Y 375.973,Z 671.465,A -85,B 0,C 180,E1 -12278.272,E2 -12278.272} C_VEL
LIN {X 0,Y 375.984,Z 671.438,A -85,B 0,C 180,E1 -12281.611,E2 -12281.611} C_VEL
LIN {X 0,Y 375.966,Z 671.444,A -85,B 0,C 180,E1 -12285.263,E2 -12285.263} C_VEL
LIN {X 0,Y 375.976,Z 671.694,A -85,B 0,C 180,E1 -12287.805,E2 -12287.805} C_VEL
LIN {X 0,Y 379.346,Z 683.503,A -85,B 0,C 180,E1 -12291.088,E2 -12291.088} C_VEL
LIN {X 0,Y 381.123,Z 690.141,A -85,B 0,C 180,E1 -12292.759,E2 -12292.759} C_VEL
LIN {X 0,Y 390.11,Z 707.744,A -85,B 0,C 180,E1 -12294.164,E2 -12294.164} C_VEL
LIN {X 0,Y 395.716,Z 719.768,A -85,B 0,C 180,E1 -12295.004,E2 -12295.004} C_VEL
LIN {X 0,Y 400.369,Z 739.8,A -85,B 0,C 180,E1 -12295.891,E2 -12295.891} C_VEL
LIN {X 0,Y 397.379,Z 852.876,A -85,B 0,C 180,E1 -12297.988,E2 -12297.988} C_VEL
LIN {X 0,Y 396.225,Z 894.612,A -85,B 0,C 180,E1 -12298.793,E2 -12298.793} C_VEL
LIN {X 0,Y 395.417,Z 907.017,A -85,B 0,C 180,E1 -12299.123,E2 -12299.123} C_VEL
LIN {X 0,Y 394.401,Z 919.141,A -85,B 0,C 180,E1 -12299.554,E2 -12299.554} C_VEL
LIN {X 0,Y 393.293,Z 931.516,A -85,B 0,C 180,E1 -12300.125,E2 -12300.125} C_VEL
LIN {X 0,Y 392.053,Z 942.903,A -85,B 0,C 180,E1 -12300.76,E2 -12300.76} C_VEL
LIN {X 0,Y 390.391,Z 956.14,A -85,B 0,C 180,E1 -12301.654,E2 -12301.654} C_VEL
LIN {X 0,Y 388.686,Z 968.733,A -85,B 0,C 180,E1 -12302.675,E2 -12302.675} C_VEL
LIN {X 0,Y 386.964,Z 979.879,A -85,B 0,C 180,E1 -12303.725,E2 -12303.725} C_VEL
LIN {X 0,Y 385.244,Z 990.681,A -85,B 0,C 180,E1 -12304.904,E2 -12304.904} C_VEL
LIN {X 0,Y 383.53,Z 1001.182,A -85,B 0,C 180,E1 -12306.226,E2 -12306.226} C_VEL
LIN {X 0,Y 381.962,Z 1010.454,A -85,B 0,C 180,E1 -12307.556,E2 -12307.556} C_VEL
LIN {X 0,Y 380.349,Z 1020.19,A -85,B 0,C 180,E1 -12309.164,E2 -12309.164} C_VEL
LIN {X 0,Y 378.833,Z 1029.544,A -85,B 0,C 180,E1 -12310.956,E2 -12310.956} C_VEL
LIN {X 0,Y 377.699,Z 1037.321,A -85,B 0,C 180,E1 -12312.68,E2 -12312.68} C_VEL
LIN {X 0,Y 376.673,Z 1043.75,A -85,B 0,C 180,E1 -12314.304,E2 -12314.304} C_VEL
LIN {X 0,Y 375.76,Z 1051.221,A -85,B 0,C 180,E1 -12316.551,E2 -12316.551} C_VEL
LIN {X 0,Y 375.295,Z 1055.663,A -85,B 0,C 180,E1 -12318.113,E2 -12318.113} C_VEL
LIN {X 0,Y 374.83,Z 1060.758,A -85,B 0,C 180,E1 -12320.285,E2 -12320.285} C_VEL
LIN {X 0,Y 374.626,Z 1064.754,A -85,B 0,C 180,E1 -12322.454,E2 -12322.454} C_VEL
LIN {X 0,Y 374.561,Z 1066.988,A -85,B 0,C 180,E1 -12323.963,E2 -12323.963} C_VEL
LIN {X 0,Y 374.486,Z 1068.89,A -85,B 0,C 180,E1 -12325.695,E2 -12325.695} C_VEL
LIN {X 0,Y 374.446,Z 1070.353,A -85,B 0,C 180,E1 -12327.849,E2 -12327.849} C_VEL
LIN {X 0,Y 374.55,Z 1070.842,A -85,B 0,C 180,E1 -12330,E2 -12330} C_VEL
LIN {X 0,Y 374.446,Z 1070.353,A -85,B 0,C 180,E1 -12332.151,E2 -12332.151} C_VEL
LIN {X 0,Y 374.486,Z 1068.89,A -85,B 0,C 180,E1 -12334.305,E2 -12334.305} C_VEL
LIN {X 0,Y 374.563,Z 1066.426,A -85,B 0,C 180,E1 -12336.464,E2 -12336.464} C_VEL
LIN {X 0,Y 374.763,Z 1061.846,A -85,B 0,C 180,E1 -12339.172,E2 -12339.172} C_VEL
LIN {X 0,Y 375.004,Z 1058.358,A -85,B 0,C 180,E1 -12340.801,E2 -12340.801} C_VEL
LIN {X 0,Y 375.629,Z 1052.635,A -85,B 0,C 180,E1 -12342.974,E2 -12342.974} C_VEL
LIN {X 0,Y 376.193,Z 1047.574,A -85,B 0,C 180,E1 -12344.608,E2 -12344.608} C_VEL
LIN {X 0,Y 377.307,Z 1039.542,A -85,B 0,C 180,E1 -12346.781,E2 -12346.781} C_VEL
LIN {X 0,Y 378.363,Z 1032.557,A -85,B 0,C 180,E1 -12348.407,E2 -12348.407} C_VEL
LIN {X 0,Y 379.589,Z 1024.586,A -85,B 0,C 180,E1 -12350.03,E2 -12350.03} C_VEL
LIN {X 0,Y 381.112,Z 1015.472,A -85,B 0,C 180,E1 -12351.642,E2 -12351.642} C_VEL
LIN {X 0,Y 382.721,Z 1006.23,A -85,B 0,C 180,E1 -12353.068,E2 -12353.068} C_VEL
LIN {X 0,Y 384.549,Z 995.034,A -85,B 0,C 180,E1 -12354.568,E2 -12354.568} C_VEL
LIN {X 0,Y 386.334,Z 983.618,A -85,B 0,C 180,E1 -12355.886,E2 -12355.886} C_VEL
LIN {X 0,Y 387.986,Z 973.195,A -85,B 0,C 180,E1 -12356.926,E2 -12356.926} C_VEL
LIN {X 0,Y 389.759,Z 961.17,A -85,B 0,C 180,E1 -12357.957,E2 -12357.957} C_VEL
LIN {X 0,Y 391.321,Z 948.847,A -85,B 0,C 180,E1 -12358.859,E2 -12358.859} C_VEL
LIN {X 0,Y 392.801,Z 936.302,A -85,B 0,C 180,E1 -12359.621,E2 -12359.621} C_VEL
LIN {X 0,Y 394.059,Z 922.871,A -85,B 0,C 180,E1 -12360.29,E2 -12360.29} C_VEL
LIN {X 0,Y 395.205,Z 909.955,A -85,B 0,C 180,E1 -12360.784,E2 -12360.784} C_VEL
LIN {X 0,Y 396.134,Z 896.946,A -85,B 0,C 180,E1 -12361.153,E2 -12361.153} C_VEL
LIN {X 0,Y 396.905,Z 871.092,A -85,B 0,C 180,E1 -12361.675,E2 -12361.675} C_VEL
LIN {X 0,Y 400.43,Z 740.88,A -85,B 0,C 180,E1 -12364.08,E2 -12364.08} C_VEL
LIN {X 0,Y 395.868,Z 720.141,A -85,B 0,C 180,E1 -12364.972,E2 -12364.972} C_VEL
LIN {X 0,Y 387.313,Z 702.094,A -85,B 0,C 180,E1 -12366.26,E2 -12366.26} C_VEL
LIN {X 0,Y 381.062,Z 690.052,A -85,B 0,C 180,E1 -12367.256,E2 -12367.256} C_VEL
LIN {X 0,Y 378.249,Z 679.422,A -85,B 0,C 180,E1 -12370.006,E2 -12370.006} C_VEL
LIN {X 0,Y 375.976,Z 671.675,A -85,B 0,C 180,E1 -12372.195,E2 -12372.195} C_VEL
LIN {X 0,Y 375.976,Z 671.447,A -85,B 0,C 180,E1 -12375.259,E2 -12375.259} C_VEL
LIN {X 0,Y 375.984,Z 671.438,A -85,B 0,C 180,E1 -12378.389,E2 -12378.389} C_VEL
LIN {X 0,Y 375.963,Z 671.463,A -85,B 0,C 180,E1 -12381.911,E2 -12381.911} C_VEL
LIN {X 0,Y 375.973,Z 671.44,A -85,B 0,C 180,E1 -12385.332,E2 -12385.332} C_VEL
LIN {X 0,Y 375.953,Z 671.459,A -85,B 0,C 180,E1 -12388.438,E2 -12388.438} C_VEL
LIN {X 0,Y 375.995,Z 671.414,A -85,B 0,C 180,E1 -12392.141,E2 -12392.141} C_VEL
LIN {X 0,Y 375.999,Z 671.458,A -85,B 0,C 180,E1 -12394.538,E2 -12394.538} C_VEL
LIN {X 0,Y 375.958,Z 671.453,A -85,B 0,C 180,E1 -12398.045,E2 -12398.045} C_VEL
LIN {X 0,Y 376.021,Z 671.447,A -85,B 0,C 180,E1 -12401.474,E2 -12401.474} C_VEL
LIN {X 0,Y 376.051,Z 671.455,A -85,B 0,C 180,E1 -12404.832,E2 -12404.832} C_VEL
LIN {X 0,Y 376.051,Z 671.445,A -85,B 0,C 180,E1 -12408.136,E2 -12408.136} C_VEL
LIN {X 0,Y 376.212,Z 671.414,A -85,B 0,C 180,E1 -12411.917,E2 -12411.917} C_VEL
LIN {X 0,Y 376.169,Z 671.437,A -85,B 0,C 180,E1 -12414.64,E2 -12414.64} C_VEL
LIN {X 0,Y 376.345,Z 671.404,A -85,B 0,C 180,E1 -12417.859,E2 -12417.859} C_VEL
LIN {X 0,Y 376.481,Z 671.399,A -85,B 0,C 180,E1 -12420,E2 -12420} C_VEL
LIN {X 0,Y 376.183,Z 671.422,A -85,B 0,C 180,E1 -12423.213,E2 -12423.213} C_VEL
LIN {X 0,Y 376.227,Z 671.424,A -85,B 0,C 180,E1 -12426.555,E2 -12426.555} C_VEL
LIN {X 0,Y 376.112,Z 671.445,A -85,B 0,C 180,E1 -12429.681,E2 -12429.681} C_VEL
LIN {X 0,Y 376.08,Z 671.436,A -85,B 0,C 180,E1 -12433.657,E2 -12433.657} C_VEL
LIN {X 0,Y 376.035,Z 671.442,A -85,B 0,C 180,E1 -12437.608,E2 -12437.608} C_VEL
LIN {X 0,Y 375.997,Z 671.457,A -85,B 0,C 180,E1 -12440.844,E2 -12440.844} C_VEL
LIN {X 0,Y 375.989,Z 671.463,A -85,B 0,C 180,E1 -12444.281,E2 -12444.281} C_VEL
LIN {X 0,Y 376.011,Z 671.437,A -85,B 0,C 180,E1 -12446.652,E2 -12446.652} C_VEL
LIN {X 0,Y 375.967,Z 671.415,A -85,B 0,C 180,E1 -12449.079,E2 -12449.079} C_VEL
LIN {X 0,Y 375.941,Z 671.47,A -85,B 0,C 180,E1 -12452.829,E2 -12452.829} C_VEL
LIN {X 0,Y 375.949,Z 671.428,A -85,B 0,C 180,E1 -12455.416,E2 -12455.416} C_VEL
LIN {X 0,Y 375.97,Z 671.454,A -85,B 0,C 180,E1 -12458.272,E2 -12458.272} C_VEL
LIN {X 0,Y 375.982,Z 671.465,A -85,B 0,C 180,E1 -12461.611,E2 -12461.611} C_VEL
LIN {X 0,Y 375.962,Z 671.468,A -85,B 0,C 180,E1 -12465.262,E2 -12465.262} C_VEL
LIN {X 0,Y 375.974,Z 671.465,A -85,B 0,C 180,E1 -12469.139,E2 -12469.139} C_VEL
LIN {X 0,Y 375.961,Z 671.467,A -85,B 0,C 180,E1 -12471.912,E2 -12471.912} C_VEL
LIN {X 0,Y 375.974,Z 671.466,A -85,B 0,C 180,E1 -12475.333,E2 -12475.333} C_VEL
LIN {X 0,Y 375.954,Z 671.467,A -85,B 0,C 180,E1 -12478.439,E2 -12478.439} C_VEL
LIN {X 0,Y 375.997,Z 671.463,A -85,B 0,C 180,E1 -12482.142,E2 -12482.142} C_VEL
LIN {X 0,Y 376.001,Z 671.463,A -85,B 0,C 180,E1 -12484.539,E2 -12484.539} C_VEL
LIN {X 0,Y 376.012,Z 671.625,A -85,B 0,C 180,E1 -12486.751,E2 -12486.751} C_VEL
LIN {X 0,Y 376.286,Z 672.855,A -85,B 0,C 180,E1 -12487.488,E2 -12487.488} C_VEL
LIN {X 0,Y 377.564,Z 675.174,A -85,B 0,C 180,E1 -12488.431,E2 -12488.431} C_VEL
LIN {X 0,Y 379.932,Z 676.995,A -85,B 0,C 180,E1 -12489.989,E2 -12489.989} C_VEL
LIN {X 0,Y 381.666,Z 678.09,A -85,B 0,C 180,E1 -12491.202,E2 -12491.202} C_VEL
LIN {X 0,Y 383.658,Z 681.241,A -85,B 0,C 180,E1 -12492.836,E2 -12492.836} C_VEL
LIN {X 0,Y 385.774,Z 682.943,A -85,B 0,C 180,E1 -12494.629,E2 -12494.629} C_VEL
LIN {X 0,Y 387.8,Z 684.122,A -85,B 0,C 180,E1 -12496.471,E2 -12496.471} C_VEL
LIN {X 0,Y 389.559,Z 687.012,A -85,B 0,C 180,E1 -12498.554,E2 -12498.554} C_VEL
LIN {X 0,Y 391.033,Z 688.471,A -85,B 0,C 180,E1 -12500.467,E2 -12500.467} C_VEL
LIN {X 0,Y 392.529,Z 689.287,A -85,B 0,C 180,E1 -12502.8,E2 -12502.8} C_VEL
LIN {X 0,Y 393.749,Z 690.02,A -85,B 0,C 180,E1 -12505.504,E2 -12505.504} C_VEL
LIN {X 0,Y 394.381,Z 690.285,A -85,B 0,C 180,E1 -12507.958,E2 -12507.958} C_VEL
LIN {X 0,Y 394.586,Z 690.322,A -85,B 0,C 180,E1 -12510,E2 -12510} C_VEL
LIN {X 0,Y 394.381,Z 690.286,A -85,B 0,C 180,E1 -12512.042,E2 -12512.042} C_VEL
LIN {X 0,Y 393.748,Z 690.015,A -85,B 0,C 180,E1 -12514.495,E2 -12514.495} C_VEL
LIN {X 0,Y 392.529,Z 689.288,A -85,B 0,C 180,E1 -12517.2,E2 -12517.2} C_VEL
LIN {X 0,Y 390.873,Z 688.355,A -85,B 0,C 180,E1 -12519.743,E2 -12519.743} C_VEL
LIN {X 0,Y 389.357,Z 686.755,A -85,B 0,C 180,E1 -12521.716,E2 -12521.716} C_VEL
LIN {X 0,Y 387.694,Z 684.018,A -85,B 0,C 180,E1 -12523.63,E2 -12523.63} C_VEL
LIN {X 0,Y 384.654,Z 682.194,A -85,B 0,C 180,E1 -12526.314,E2 -12526.314} C_VEL
LIN {X 0,Y 382.88,Z 680.219,A -85,B 0,C 180,E1 -12527.78,E2 -12527.78} C_VEL
LIN {X 0,Y 381.459,Z 677.86,A -85,B 0,C 180,E1 -12528.948,E2 -12528.948} C_VEL
LIN {X 0,Y 377.914,Z 675.556,A -85,B 0,C 180,E1 -12531.349,E2 -12531.349} C_VEL
LIN {X 0,Y 376.362,Z 673.138,A -85,B 0,C 180,E1 -12532.435,E2 -12532.435} C_VEL
LIN {X 0,Y 376.064,Z 671.936,A -85,B 0,C 180,E1 -12532.961,E2 -12532.961} C_VEL
LIN {X 0,Y 375.991,Z 671.496,A -85,B 0,C 180,E1 -12533.667,E2 -12533.667} C_VEL
LIN {X 0,Y 376.014,Z 671.462,A -85,B 0,C 180,E1 -12536.652,E2 -12536.652} C_VEL
LIN {X 0,Y 375.971,Z 671.465,A -85,B 0,C 180,E1 -12539.078,E2 -12539.078} C_VEL
LIN {X 0,Y 375.943,Z 671.468,A -85,B 0,C 180,E1 -12542.828,E2 -12542.828} C_VEL
LIN {X 0,Y 375.952,Z 671.467,A -85,B 0,C 180,E1 -12545.415,E2 -12545.415} C_VEL
LIN {X 0,Y 375.971,Z 671.465,A -85,B 0,C 180,E1 -12548.271,E2 -12548.271} C_VEL
LIN {X 0,Y 375.986,Z 671.462,A -85,B 0,C 180,E1 -12550.038,E2 -12550.038} C_VEL
LIN {X 0,Y 375.274,Z 671.553,A -85,B 0,C 180,E1 -12550.931,E2 -12550.931} C_VEL
LIN {X 0,Y 372.37,Z 671.914,A -85,B 0,C 180,E1 -12552.384,E2 -12552.384} C_VEL
LIN {X 0,Y 369.961,Z 672.214,A -85,B 0,C 180,E1 -12553.558,E2 -12553.558} C_VEL
LIN {X 0,Y 368.971,Z 672.339,A -85,B 0,C 180,E1 -12554.467,E2 -12554.467} C_VEL
LIN {X 0,Y 368.912,Z 672.346,A -85,B 0,C 180,E1 -12554.774,E2 -12554.774} C_VEL
LIN {X 0,Y 368.933,Z 672.343,A -85,B 0,C 180,E1 -12558.185,E2 -12558.185} C_VEL
LIN {X 0,Y 368.905,Z 672.339,A -85,B 0,C 180,E1 -12561.358,E2 -12561.358} C_VEL
LIN {X 0,Y 368.928,Z 672.31,A -85,B 0,C 180,E1 -12565.146,E2 -12565.146} C_VEL
LIN {X 0,Y 368.921,Z 672.323,A -85,B 0,C 180,E1 -12569.046,E2 -12569.046} C_VEL
LIN {X 0,Y 368.977,Z 672.284,A -85,B 0,C 180,E1 -12571.564,E2 -12571.564} C_VEL
LIN {X 0,Y 368.951,Z 672.339,A -85,B 0,C 180,E1 -12575.225,E2 -12575.225} C_VEL
LIN {X 0,Y 368.962,Z 672.333,A -85,B 0,C 180,E1 -12578.959,E2 -12578.959} C_VEL
LIN {X 0,Y 368.982,Z 672.319,A -85,B 0,C 180,E1 -12582.257,E2 -12582.257} C_VEL
LIN {X 0,Y 369.028,Z 672.315,A -85,B 0,C 180,E1 -12586.228,E2 -12586.228} C_VEL
LIN {X 0,Y 369.06,Z 672.324,A -85,B 0,C 180,E1 -12590.132,E2 -12590.132} C_VEL
LIN {X 0,Y 369.152,Z 672.297,A -85,B 0,C 180,E1 -12592.342,E2 -12592.342} C_VEL
LIN {X 0,Y 369.141,Z 672.316,A -85,B 0,C 180,E1 -12594.538,E2 -12594.538} C_VEL
LIN {X 0,Y 369.31,Z 672.275,A -85,B 0,C 180,E1 -12597.819,E2 -12597.819} C_VEL
LIN {X 0,Y 369.45,Z 672.276,A -85,B 0,C 180,E1 -12600,E2 -12600} C_VEL
LIN {X 0,Y 369.31,Z 672.281,A -85,B 0,C 180,E1 -12602.181,E2 -12602.181} C_VEL
LIN {X 0,Y 369.2,Z 672.3,A -85,B 0,C 180,E1 -12606.559,E2 -12606.559} C_VEL
LIN {X 0,Y 369.114,Z 672.301,A -85,B 0,C 180,E1 -12608.762,E2 -12608.762} C_VEL
LIN {X 0,Y 369.005,Z 672.321,A -85,B 0,C 180,E1 -12612.093,E2 -12612.093} C_VEL
LIN {X 0,Y 368.99,Z 672.334,A -85,B 0,C 180,E1 -12615.465,E2 -12615.465} C_VEL
LIN {X 0,Y 368.981,Z 672.326,A -85,B 0,C 180,E1 -12618.893,E2 -12618.893} C_VEL
LIN {X 0,Y 368.926,Z 672.326,A -85,B 0,C 180,E1 -12622.396,E2 -12622.396} C_VEL
LIN {X 0,Y 368.992,Z 672.323,A -85,B 0,C 180,E1 -12625.981,E2 -12625.981} C_VEL
LIN {X 0,Y 368.96,Z 672.282,A -85,B 0,C 180,E1 -12628.814,E2 -12628.814} C_VEL
LIN {X 0,Y 368.892,Z 672.348,A -85,B 0,C 180,E1 -12632.239,E2 -12632.239} C_VEL
LIN {X 0,Y 368.923,Z 672.313,A -85,B 0,C 180,E1 -12635.002,E2 -12635.002} C_VEL
LIN {X 0,Y 368.909,Z 672.346,A -85,B 0,C 180,E1 -12638.642,E2 -12638.642} C_VEL
LIN {X 0,Y 368.937,Z 672.319,A -85,B 0,C 180,E1 -12642.021,E2 -12642.021} C_VEL
LIN {X 0,Y 368.92,Z 672.322,A -85,B 0,C 180,E1 -12645.184,E2 -12645.184} C_VEL
LIN {X 0,Y 368.916,Z 672.425,A -85,B 0,C 180,E1 -12647.021,E2 -12647.021} C_VEL
LIN {X 0,Y 370.764,Z 678.812,A -85,B 0,C 180,E1 -12648.94,E2 -12648.94} C_VEL
LIN {X 0,Y 373.711,Z 689.588,A -85,B 0,C 180,E1 -12651.86,E2 -12651.86} C_VEL
LIN {X 0,Y 377.556,Z 697.087,A -85,B 0,C 180,E1 -12652.537,E2 -12652.537} C_VEL
LIN {X 0,Y 385.33,Z 712.284,A -85,B 0,C 180,E1 -12653.755,E2 -12653.755} C_VEL
LIN {X 0,Y 390.431,Z 723.529,A -85,B 0,C 180,E1 -12654.547,E2 -12654.547} C_VEL
LIN {X 0,Y 394.506,Z 741.472,A -85,B 0,C 180,E1 -12655.353,E2 -12655.353} C_VEL
LIN {X 0,Y 390.207,Z 893.373,A -85,B 0,C 180,E1 -12658.228,E2 -12658.228} C_VEL
LIN {X 0,Y 389.41,Z 905.832,A -85,B 0,C 180,E1 -12658.555,E2 -12658.555} C_VEL
LIN {X 0,Y 388.302,Z 918.935,A -85,B 0,C 180,E1 -12659.024,E2 -12659.024} C_VEL
LIN {X 0,Y 387.118,Z 931.309,A -85,B 0,C 180,E1 -12659.599,E2 -12659.599} C_VEL
LIN {X 0,Y 385.851,Z 942.697,A -85,B 0,C 180,E1 -12660.243,E2 -12660.243} C_VEL
LIN {X 0,Y 384.111,Z 955.933,A -85,B 0,C 180,E1 -12661.147,E2 -12661.147} C_VEL
LIN {X 0,Y 382.521,Z 967.353,A -85,B 0,C 180,E1 -12662.076,E2 -12662.076} C_VEL
LIN {X 0,Y 380.517,Z 979.67,A -85,B 0,C 180,E1 -12663.245,E2 -12663.245} C_VEL
LIN {X 0,Y 378.781,Z 990.474,A -85,B 0,C 180,E1 -12664.445,E2 -12664.445} C_VEL
LIN {X 0,Y 376.945,Z 1000.974,A -85,B 0,C 180,E1 -12665.784,E2 -12665.784} C_VEL
LIN {X 0,Y 375.322,Z 1010.246,A -85,B 0,C 180,E1 -12667.136,E2 -12667.136} C_VEL
LIN {X 0,Y 373.625,Z 1019.982,A -85,B 0,C 180,E1 -12668.771,E2 -12668.771} C_VEL
LIN {X 0,Y 372.135,Z 1028.558,A -85,B 0,C 180,E1 -12670.426,E2 -12670.426} C_VEL
LIN {X 0,Y 370.785,Z 1037.111,A -85,B 0,C 180,E1 -12672.346,E2 -12672.346} C_VEL
LIN {X 0,Y 369.724,Z 1043.541,A -85,B 0,C 180,E1 -12674.001,E2 -12674.001} C_VEL
LIN {X 0,Y 368.81,Z 1050.617,A -85,B 0,C 180,E1 -12676.155,E2 -12676.155} C_VEL
LIN {X 0,Y 368.258,Z 1055.455,A -85,B 0,C 180,E1 -12677.882,E2 -12677.882} C_VEL
LIN {X 0,Y 367.748,Z 1060.55,A -85,B 0,C 180,E1 -12680.096,E2 -12680.096} C_VEL
LIN {X 0,Y 367.544,Z 1064.547,A -85,B 0,C 180,E1 -12682.308,E2 -12682.308} C_VEL
LIN {X 0,Y 367.476,Z 1066.935,A -85,B 0,C 180,E1 -12683.989,E2 -12683.989} C_VEL
LIN {X 0,Y 367.395,Z 1068.684,A -85,B 0,C 180,E1 -12685.612,E2 -12685.612} C_VEL
LIN {X 0,Y 367.346,Z 1070.148,A -85,B 0,C 180,E1 -12687.807,E2 -12687.807} C_VEL
LIN {X 0,Y 367.453,Z 1070.637,A -85,B 0,C 180,E1 -12690,E2 -12690} C_VEL
LIN {X 0,Y 367.346,Z 1070.148,A -85,B 0,C 180,E1 -12692.193,E2 -12692.193} C_VEL
LIN {X 0,Y 367.395,Z 1068.684,A -85,B 0,C 180,E1 -12694.388,E2 -12694.388} C_VEL
LIN {X 0,Y 367.478,Z 1066.22,A -85,B 0,C 180,E1 -12696.589,E2 -12696.589} C_VEL
LIN {X 0,Y 367.691,Z 1061.638,A -85,B 0,C 180,E1 -12699.35,E2 -12699.35} C_VEL
LIN {X 0,Y 367.978,Z 1058.151,A -85,B 0,C 180,E1 -12701.01,E2 -12701.01} C_VEL
LIN {X 0,Y 368.616,Z 1052.427,A -85,B 0,C 180,E1 -12703.226,E2 -12703.226} C_VEL
LIN {X 0,Y 369.223,Z 1047.365,A -85,B 0,C 180,E1 -12704.89,E2 -12704.89} C_VEL
LIN {X 0,Y 370.44,Z 1039.334,A -85,B 0,C 180,E1 -12707.101,E2 -12707.101} C_VEL
LIN {X 0,Y 371.528,Z 1032.349,A -85,B 0,C 180,E1 -12708.758,E2 -12708.758} C_VEL
LIN {X 0,Y 372.828,Z 1024.378,A -85,B 0,C 180,E1 -12710.409,E2 -12710.409} C_VEL
LIN {X 0,Y 374.408,Z 1015.263,A -85,B 0,C 180,E1 -12712.05,E2 -12712.05} C_VEL
LIN {X 0,Y 376.287,Z 1005.019,A -85,B 0,C 180,E1 -12713.64,E2 -12713.64} C_VEL
LIN {X 0,Y 377.99,Z 994.825,A -85,B 0,C 180,E1 -12715.023,E2 -12715.023} C_VEL
LIN {X 0,Y 379.686,Z 984.658,A -85,B 0,C 180,E1 -12716.226,E2 -12716.226} C_VEL
LIN {X 0,Y 381.627,Z 972.989,A -85,B 0,C 180,E1 -12717.412,E2 -12717.412} C_VEL
LIN {X 0,Y 383.451,Z 960.962,A -85,B 0,C 180,E1 -12718.459,E2 -12718.459} C_VEL
LIN {X 0,Y 385.074,Z 948.64,A -85,B 0,C 180,E1 -12719.372,E2 -12719.372} C_VEL
LIN {X 0,Y 386.633,Z 936.096,A -85,B 0,C 180,E1 -12720.142,E2 -12720.142} C_VEL
LIN {X 0,Y 387.928,Z 922.665,A -85,B 0,C 180,E1 -12720.821,E2 -12720.821} C_VEL
LIN {X 0,Y 389.126,Z 909.75,A -85,B 0,C 180,E1 -12721.319,E2 -12721.319} C_VEL
LIN {X 0,Y 390.101,Z 896.338,A -85,B 0,C 180,E1 -12721.701,E2 -12721.701} C_VEL
LIN {X 0,Y 390.884,Z 870.026,A -85,B 0,C 180,E1 -12722.24,E2 -12722.24} C_VEL
LIN {X 0,Y 394.44,Z 741.338,A -85,B 0,C 180,E1 -12724.657,E2 -12724.657} C_VEL
LIN {X 0,Y 390.176,Z 722.712,A -85,B 0,C 180,E1 -12725.498,E2 -12725.498} C_VEL
LIN {X 0,Y 380.856,Z 703.136,A -85,B 0,C 180,E1 -12726.947,E2 -12726.947} C_VEL
LIN {X 0,Y 373.786,Z 689.71,A -85,B 0,C 180,E1 -12728.114,E2 -12728.114} C_VEL
LIN {X 0,Y 371.11,Z 679.873,A -85,B 0,C 180,E1 -12730.755,E2 -12730.755} C_VEL
LIN {X 0,Y 368.944,Z 672.587,A -85,B 0,C 180,E1 -12732.887,E2 -12732.887} C_VEL
LIN {X 0,Y 368.92,Z 672.322,A -85,B 0,C 180,E1 -12734.816,E2 -12734.816} C_VEL
LIN {X 0,Y 368.936,Z 672.317,A -85,B 0,C 180,E1 -12738.185,E2 -12738.185} C_VEL
LIN {X 0,Y 368.909,Z 672.346,A -85,B 0,C 180,E1 -12741.358,E2 -12741.358} C_VEL
LIN {X 0,Y 368.93,Z 672.314,A -85,B 0,C 180,E1 -12745.146,E2 -12745.146} C_VEL
LIN {X 0,Y 368.923,Z 672.32,A -85,B 0,C 180,E1 -12749.046,E2 -12749.046} C_VEL
LIN {X 0,Y 368.979,Z 672.281,A -85,B 0,C 180,E1 -12751.564,E2 -12751.564} C_VEL
LIN {X 0,Y 368.95,Z 672.339,A -85,B 0,C 180,E1 -12755.224,E2 -12755.224} C_VEL
LIN {X 0,Y 368.962,Z 672.336,A -85,B 0,C 180,E1 -12758.959,E2 -12758.959} C_VEL
LIN {X 0,Y 368.983,Z 672.321,A -85,B 0,C 180,E1 -12762.257,E2 -12762.257} C_VEL
LIN {X 0,Y 369.029,Z 672.318,A -85,B 0,C 180,E1 -12766.227,E2 -12766.227} C_VEL
LIN {X 0,Y 369.064,Z 672.322,A -85,B 0,C 180,E1 -12770.131,E2 -12770.131} C_VEL
LIN {X 0,Y 369.156,Z 672.293,A -85,B 0,C 180,E1 -12772.341,E2 -12772.341} C_VEL
LIN {X 0,Y 369.141,Z 672.312,A -85,B 0,C 180,E1 -12774.537,E2 -12774.537} C_VEL
LIN {X 0,Y 369.31,Z 672.279,A -85,B 0,C 180,E1 -12777.819,E2 -12777.819} C_VEL
LIN {X 0,Y 369.45,Z 672.275,A -85,B 0,C 180,E1 -12780,E2 -12780} C_VEL
LIN {X 0,Y 369.31,Z 672.274,A -85,B 0,C 180,E1 -12782.181,E2 -12782.181} C_VEL
LIN {X 0,Y 369.197,Z 672.301,A -85,B 0,C 180,E1 -12786.558,E2 -12786.558} C_VEL
LIN {X 0,Y 369.113,Z 672.31,A -85,B 0,C 180,E1 -12788.761,E2 -12788.761} C_VEL
LIN {X 0,Y 368.996,Z 672.317,A -85,B 0,C 180,E1 -12792.093,E2 -12792.093} C_VEL
LIN {X 0,Y 368.988,Z 672.333,A -85,B 0,C 180,E1 -12795.465,E2 -12795.465} C_VEL
LIN {X 0,Y 368.984,Z 672.33,A -85,B 0,C 180,E1 -12798.892,E2 -12798.892} C_VEL
LIN {X 0,Y 368.948,Z 672.327,A -85,B 0,C 180,E1 -12802.394,E2 -12802.394} C_VEL
LIN {X 0,Y 368.991,Z 672.321,A -85,B 0,C 180,E1 -12805.98,E2 -12805.98} C_VEL
LIN {X 0,Y 368.958,Z 672.286,A -85,B 0,C 180,E1 -12808.813,E2 -12808.813} C_VEL
LIN {X 0,Y 368.89,Z 672.346,A -85,B 0,C 180,E1 -12812.238,E2 -12812.238} C_VEL
LIN {X 0,Y 368.921,Z 672.308,A -85,B 0,C 180,E1 -12815.002,E2 -12815.002} C_VEL
LIN {X 0,Y 368.905,Z 672.339,A -85,B 0,C 180,E1 -12818.642,E2 -12818.642} C_VEL
LIN {X 0,Y 368.934,Z 672.342,A -85,B 0,C 180,E1 -12822.02,E2 -12822.02} C_VEL
LIN {X 0,Y 368.916,Z 672.346,A -85,B 0,C 180,E1 -12825.183,E2 -12825.183} C_VEL
LIN {X 0,Y 368.903,Z 672.346,A -85,B 0,C 180,E1 -12828.182,E2 -12828.182} C_VEL
LIN {X 0,Y 368.906,Z 672.345,A -85,B 0,C 180,E1 -12831.359,E2 -12831.359} C_VEL
LIN {X 0,Y 368.93,Z 672.344,A -85,B 0,C 180,E1 -12835.147,E2 -12835.147} C_VEL
LIN {X 0,Y 368.923,Z 672.344,A -85,B 0,C 180,E1 -12839.047,E2 -12839.047} C_VEL
LIN {X 0,Y 368.981,Z 672.336,A -85,B 0,C 180,E1 -12841.565,E2 -12841.565} C_VEL
LIN {X 0,Y 368.987,Z 672.536,A -85,B 0,C 180,E1 -12843.223,E2 -12843.223} C_VEL
LIN {X 0,Y 369.3,Z 673.715,A -85,B 0,C 180,E1 -12843.903,E2 -12843.903} C_VEL
LIN {X 0,Y 370.676,Z 676.155,A -85,B 0,C 180,E1 -12844.749,E2 -12844.749} C_VEL
LIN {X 0,Y 373.121,Z 677.981,A -85,B 0,C 180,E1 -12846.14,E2 -12846.14} C_VEL
LIN {X 0,Y 374.436,Z 678.892,A -85,B 0,C 180,E1 -12846.933,E2 -12846.933} C_VEL
LIN {X 0,Y 376.235,Z 681.922,A -85,B 0,C 180,E1 -12848.163,E2 -12848.163} C_VEL
LIN {X 0,Y 378.373,Z 683.674,A -85,B 0,C 180,E1 -12849.564,E2 -12849.564} C_VEL
LIN {X 0,Y 380.482,Z 684.969,A -85,B 0,C 180,E1 -12851.001,E2 -12851.001} C_VEL
LIN {X 0,Y 382.537,Z 688.155,A -85,B 0,C 180,E1 -12852.663,E2 -12852.663} C_VEL
LIN {X 0,Y 384.882,Z 690.003,A -85,B 0,C 180,E1 -12854.619,E2 -12854.619} C_VEL
LIN {X 0,Y 386.882,Z 691.184,A -85,B 0,C 180,E1 -12856.438,E2 -12856.438} C_VEL
LIN {X 0,Y 388.458,Z 693.823,A -85,B 0,C 180,E1 -12858.257,E2 -12858.257} C_VEL
LIN {X 0,Y 389.891,Z 695.329,A -85,B 0,C 180,E1 -12860.113,E2 -12860.113} C_VEL
LIN {X 0,Y 391.652,Z 696.332,A -85,B 0,C 180,E1 -12862.784,E2 -12862.784} C_VEL
LIN {X 0,Y 392.878,Z 697.066,A -85,B 0,C 180,E1 -12865.494,E2 -12865.494} C_VEL
LIN {X 0,Y 393.518,Z 697.315,A -85,B 0,C 180,E1 -12867.953,E2 -12867.953} C_VEL
LIN {X 0,Y 393.72,Z 697.37,A -85,B 0,C 180,E1 -12870,E2 -12870} C_VEL
LIN {X 0,Y 393.518,Z 697.318,A -85,B 0,C 180,E1 -12872.047,E2 -12872.047} C_VEL
LIN {X 0,Y 392.878,Z 697.062,A -85,B 0,C 180,E1 -12874.505,E2 -12874.505} C_VEL
LIN {X 0,Y 391.652,Z 696.333,A -85,B 0,C 180,E1 -12877.216,E2 -12877.216} C_VEL
LIN {X 0,Y 389.983,Z 695.403,A -85,B 0,C 180,E1 -12879.766,E2 -12879.766} C_VEL
LIN {X 0,Y 388.351,Z 693.695,A -85,B 0,C 180,E1 -12881.879,E2 -12881.879} C_VEL
LIN {X 0,Y 386.496,Z 690.799,A -85,B 0,C 180,E1 -12883.941,E2 -12883.941} C_VEL
LIN {X 0,Y 383.715,Z 689.254,A -85,B 0,C 180,E1 -12886.355,E2 -12886.355} C_VEL
LIN {X 0,Y 381.746,Z 687.136,A -85,B 0,C 180,E1 -12887.966,E2 -12887.966} C_VEL
LIN {X 0,Y 380.175,Z 684.644,A -85,B 0,C 180,E1 -12889.225,E2 -12889.225} C_VEL
LIN {X 0,Y 376.905,Z 682.635,A -85,B 0,C 180,E1 -12891.409,E2 -12891.409} C_VEL
LIN {X 0,Y 375.107,Z 680.135,A -85,B 0,C 180,E1 -12892.627,E2 -12892.627} C_VEL
LIN {X 0,Y 373.973,Z 678.409,A -85,B 0,C 180,E1 -12893.353,E2 -12893.353} C_VEL
LIN {X 0,Y 370.954,Z 676.478,A -85,B 0,C 180,E1 -12895.08,E2 -12895.08} C_VEL
LIN {X 0,Y 369.435,Z 674.115,A -85,B 0,C 180,E1 -12895.993,E2 -12895.993} C_VEL
LIN {X 0,Y 369.063,Z 672.875,A -85,B 0,C 180,E1 -12896.492,E2 -12896.492} C_VEL
LIN {X 0,Y 368.966,Z 672.366,A -85,B 0,C 180,E1 -12897.202,E2 -12897.202} C_VEL
LIN {X 0,Y 368.918,Z 672.345,A -85,B 0,C 180,E1 -12899.689,E2 -12899.689} C_VEL
LIN {X 0,Y 368.89,Z 672.349,A -85,B 0,C 180,E1 -12903.538,E2 -12903.538} C_VEL
LIN {X 0,Y 368.897,Z 672.346,A -85,B 0,C 180,E1 -12906.856,E2 -12906.856} C_VEL
LIN {X 0,Y 368.946,Z 672.341,A -85,B 0,C 180,E1 -12910.364,E2 -12910.364} C_VEL
LIN {X 0,Y 368.892,Z 672.347,A -85,B 0,C 180,E1 -12913.618,E2 -12913.618} C_VEL
LIN {X 0,Y 368.912,Z 672.346,A -85,B 0,C 180,E1 -12914.774,E2 -12914.774} C_VEL
LIN {X 0,Y 368.306,Z 672.427,A -85,B 0,C 180,E1 -12915.685,E2 -12915.685} C_VEL
LIN {X 0,Y 365.476,Z 672.781,A -85,B 0,C 180,E1 -12917.167,E2 -12917.167} C_VEL
LIN {X 0,Y 363.033,Z 673.081,A -85,B 0,C 180,E1 -12918.365,E2 -12918.365} C_VEL
LIN {X 0,Y 361.969,Z 673.211,A -85,B 0,C 180,E1 -12919.292,E2 -12919.292} C_VEL
LIN {X 0,Y 361.876,Z 673.22,A -85,B 0,C 180,E1 -12919.606,E2 -12919.606} C_VEL
LIN {X 0,Y 361.861,Z 673.182,A -85,B 0,C 180,E1 -12922.982,E2 -12922.982} C_VEL
LIN {X 0,Y 361.85,Z 673.221,A -85,B 0,C 180,E1 -12926.63,E2 -12926.63} C_VEL
LIN {X 0,Y 361.867,Z 673.185,A -85,B 0,C 180,E1 -12929.672,E2 -12929.672} C_VEL
LIN {X 0,Y 361.946,Z 673.189,A -85,B 0,C 180,E1 -12933.475,E2 -12933.475} C_VEL
LIN {X 0,Y 361.9,Z 673.206,A -85,B 0,C 180,E1 -12937.146,E2 -12937.146} C_VEL
LIN {X 0,Y 361.924,Z 673.211,A -85,B 0,C 180,E1 -12940.725,E2 -12940.725} C_VEL
LIN {X 0,Y 361.936,Z 673.212,A -85,B 0,C 180,E1 -12944.226,E2 -12944.226} C_VEL
LIN {X 0,Y 361.989,Z 673.188,A -85,B 0,C 180,E1 -12946.528,E2 -12946.528} C_VEL
LIN {X 0,Y 362.024,Z 673.201,A -85,B 0,C 180,E1 -12949.938,E2 -12949.938} C_VEL
LIN {X 0,Y 362.157,Z 673.175,A -85,B 0,C 180,E1 -12953.314,E2 -12953.314} C_VEL
LIN {X 0,Y 362.274,Z 673.151,A -85,B 0,C 180,E1 -12957.777,E2 -12957.777} C_VEL
LIN {X 0,Y 362.42,Z 673.152,A -85,B 0,C 180,E1 -12960,E2 -12960} C_VEL
LIN {X 0,Y 362.274,Z 673.156,A -85,B 0,C 180,E1 -12962.224,E2 -12962.224} C_VEL
LIN {X 0,Y 362.16,Z 673.174,A -85,B 0,C 180,E1 -12966.687,E2 -12966.687} C_VEL
LIN {X 0,Y 362.028,Z 673.197,A -85,B 0,C 180,E1 -12970.062,E2 -12970.062} C_VEL
LIN {X 0,Y 361.99,Z 673.194,A -85,B 0,C 180,E1 -12973.9,E2 -12973.9} C_VEL
LIN {X 0,Y 361.96,Z 673.194,A -85,B 0,C 180,E1 -12977.939,E2 -12977.939} C_VEL
LIN {X 0,Y 361.89,Z 673.207,A -85,B 0,C 180,E1 -12981.653,E2 -12981.653} C_VEL
LIN {X 0,Y 361.921,Z 673.214,A -85,B 0,C 180,E1 -12985.291,E2 -12985.291} C_VEL
LIN {X 0,Y 361.915,Z 673.165,A -85,B 0,C 180,E1 -12987.779,E2 -12987.779} C_VEL
LIN {X 0,Y 361.84,Z 673.211,A -85,B 0,C 180,E1 -12991.286,E2 -12991.286} C_VEL
LIN {X 0,Y 361.848,Z 673.204,A -85,B 0,C 180,E1 -12994.281,E2 -12994.281} C_VEL
LIN {X 0,Y 361.866,Z 673.201,A -85,B 0,C 180,E1 -12997.225,E2 -12997.225} C_VEL
LIN {X 0,Y 361.9,Z 673.19,A -85,B 0,C 180,E1 -13000.769,E2 -13000.769} C_VEL
LIN {X 0,Y 361.907,Z 673.203,A -85,B 0,C 180,E1 -13004.355,E2 -13004.355} C_VEL
LIN {X 0,Y 361.862,Z 673.37,A -85,B 0,C 180,E1 -13006.317,E2 -13006.317} C_VEL
LIN {X 0,Y 364.966,Z 684.034,A -85,B 0,C 180,E1 -13009.519,E2 -13009.519} C_VEL
LIN {X 0,Y 366.483,Z 689.47,A -85,B 0,C 180,E1 -13010.991,E2 -13010.991} C_VEL
LIN {X 0,Y 376.386,Z 708.295,A -85,B 0,C 180,E1 -13012.665,E2 -13012.665} C_VEL
LIN {X 0,Y 384.813,Z 725.882,A -85,B 0,C 180,E1 -13014.006,E2 -13014.006} C_VEL
LIN {X 0,Y 388.555,Z 742.506,A -85,B 0,C 180,E1 -13014.772,E2 -13014.772} C_VEL
LIN {X 0,Y 386.139,Z 825.895,A -85,B 0,C 180,E1 -13016.36,E2 -13016.36} C_VEL
LIN {X 0,Y 384.162,Z 893.736,A -85,B 0,C 180,E1 -13017.684,E2 -13017.684} C_VEL
LIN {X 0,Y 383.371,Z 905.627,A -85,B 0,C 180,E1 -13018.001,E2 -13018.001} C_VEL
LIN {X 0,Y 382.184,Z 918.728,A -85,B 0,C 180,E1 -13018.471,E2 -13018.471} C_VEL
LIN {X 0,Y 381.001,Z 931.103,A -85,B 0,C 180,E1 -13019.058,E2 -13019.058} C_VEL
LIN {X 0,Y 379.67,Z 942.49,A -85,B 0,C 180,E1 -13019.708,E2 -13019.708} C_VEL
LIN {X 0,Y 377.878,Z 955.727,A -85,B 0,C 180,E1 -13020.625,E2 -13020.625} C_VEL
LIN {X 0,Y 376.113,Z 967.775,A -85,B 0,C 180,E1 -13021.623,E2 -13021.623} C_VEL
LIN {X 0,Y 374.149,Z 979.463,A -85,B 0,C 180,E1 -13022.752,E2 -13022.752} C_VEL
LIN {X 0,Y 372.324,Z 990.266,A -85,B 0,C 180,E1 -13023.969,E2 -13023.969} C_VEL
LIN {X 0,Y 370.37,Z 1000.765,A -85,B 0,C 180,E1 -13025.326,E2 -13025.326} C_VEL
LIN {X 0,Y 368.688,Z 1010.038,A -85,B 0,C 180,E1 -13026.701,E2 -13026.701} C_VEL
LIN {X 0,Y 366.902,Z 1019.773,A -85,B 0,C 180,E1 -13028.363,E2 -13028.363} C_VEL
LIN {X 0,Y 365.325,Z 1028.299,A -85,B 0,C 180,E1 -13030.035,E2 -13030.035} C_VEL
LIN {X 0,Y 363.911,Z 1036.902,A -85,B 0,C 180,E1 -13032.002,E2 -13032.002} C_VEL
LIN {X 0,Y 362.804,Z 1043.332,A -85,B 0,C 180,E1 -13033.687,E2 -13033.687} C_VEL
LIN {X 0,Y 361.772,Z 1050.758,A -85,B 0,C 180,E1 -13036.004,E2 -13036.004} C_VEL
LIN {X 0,Y 361.233,Z 1055.247,A -85,B 0,C 180,E1 -13037.643,E2 -13037.643} C_VEL
LIN {X 0,Y 360.678,Z 1060.342,A -85,B 0,C 180,E1 -13039.9,E2 -13039.9} C_VEL
LIN {X 0,Y 360.461,Z 1064.341,A -85,B 0,C 180,E1 -13042.156,E2 -13042.156} C_VEL
LIN {X 0,Y 360.331,Z 1067.293,A -85,B 0,C 180,E1 -13044.404,E2 -13044.404} C_VEL
LIN {X 0,Y 360.308,Z 1068.478,A -85,B 0,C 180,E1 -13045.525,E2 -13045.525} C_VEL
LIN {X 0,Y 360.251,Z 1069.942,A -85,B 0,C 180,E1 -13047.764,E2 -13047.764} C_VEL
LIN {X 0,Y 360.356,Z 1070.431,A -85,B 0,C 180,E1 -13050,E2 -13050} C_VEL
LIN {X 0,Y 360.251,Z 1069.942,A -85,B 0,C 180,E1 -13052.236,E2 -13052.236} C_VEL
LIN {X 0,Y 360.308,Z 1068.478,A -85,B 0,C 180,E1 -13054.475,E2 -13054.475} C_VEL
LIN {X 0,Y 360.382,Z 1066.013,A -85,B 0,C 180,E1 -13056.719,E2 -13056.719} C_VEL
LIN {X 0,Y 360.609,Z 1061.431,A -85,B 0,C 180,E1 -13059.535,E2 -13059.535} C_VEL
LIN {X 0,Y 360.955,Z 1057.944,A -85,B 0,C 180,E1 -13061.227,E2 -13061.227} C_VEL
LIN {X 0,Y 361.627,Z 1052.219,A -85,B 0,C 180,E1 -13063.486,E2 -13063.486} C_VEL
LIN {X 0,Y 362.252,Z 1047.156,A -85,B 0,C 180,E1 -13065.183,E2 -13065.183} C_VEL
LIN {X 0,Y 363.578,Z 1039.126,A -85,B 0,C 180,E1 -13067.434,E2 -13067.434} C_VEL
LIN {X 0,Y 364.691,Z 1032.139,A -85,B 0,C 180,E1 -13069.123,E2 -13069.123} C_VEL
LIN {X 0,Y 366.093,Z 1024.169,A -85,B 0,C 180,E1 -13070.802,E2 -13070.802} C_VEL
LIN {X 0,Y 367.736,Z 1015.054,A -85,B 0,C 180,E1 -13072.471,E2 -13072.471} C_VEL
LIN {X 0,Y 369.541,Z 1005.66,A -85,B 0,C 180,E1 -13073.966,E2 -13073.966} C_VEL
LIN {X 0,Y 371.486,Z 994.617,A -85,B 0,C 180,E1 -13075.492,E2 -13075.492} C_VEL
LIN {X 0,Y 373.236,Z 984.449,A -85,B 0,C 180,E1 -13076.715,E2 -13076.715} C_VEL
LIN {X 0,Y 375.281,Z 972.781,A -85,B 0,C 180,E1 -13077.916,E2 -13077.916} C_VEL
LIN {X 0,Y 377.18,Z 960.756,A -85,B 0,C 180,E1 -13078.976,E2 -13078.976} C_VEL
LIN {X 0,Y 378.871,Z 948.434,A -85,B 0,C 180,E1 -13079.902,E2 -13079.902} C_VEL
LIN {X 0,Y 380.481,Z 935.89,A -85,B 0,C 180,E1 -13080.681,E2 -13080.681} C_VEL
LIN {X 0,Y 381.832,Z 922.459,A -85,B 0,C 180,E1 -13081.368,E2 -13081.368} C_VEL
LIN {X 0,Y 383.064,Z 909.544,A -85,B 0,C 180,E1 -13081.872,E2 -13081.872} C_VEL
LIN {X 0,Y 384.051,Z 896.543,A -85,B 0,C 180,E1 -13082.249,E2 -13082.249} C_VEL
LIN {X 0,Y 384.938,Z 868.29,A -85,B 0,C 180,E1 -13082.833,E2 -13082.833} C_VEL
LIN {X 0,Y 388.604,Z 743.768,A -85,B 0,C 180,E1 -13085.195,E2 -13085.195} C_VEL
LIN {X 0,Y 385.99,Z 730.78,A -85,B 0,C 180,E1 -13085.758,E2 -13085.758} C_VEL
LIN {X 0,Y 384.533,Z 725.451,A -85,B 0,C 180,E1 -13086.034,E2 -13086.034} C_VEL
LIN {X 0,Y 376.09,Z 707.545,A -85,B 0,C 180,E1 -13087.387,E2 -13087.387} C_VEL
LIN {X 0,Y 366.509,Z 689.424,A -85,B 0,C 180,E1 -13089.011,E2 -13089.011} C_VEL
LIN {X 0,Y 363.552,Z 679.114,A -85,B 0,C 180,E1 -13091.904,E2 -13091.904} C_VEL
LIN {X 0,Y 361.861,Z 673.373,A -85,B 0,C 180,E1 -13093.684,E2 -13093.684} C_VEL
LIN {X 0,Y 361.908,Z 673.208,A -85,B 0,C 180,E1 -13095.93,E2 -13095.93} C_VEL
LIN {X 0,Y 361.9,Z 673.19,A -85,B 0,C 180,E1 -13099.231,E2 -13099.231} C_VEL
LIN {X 0,Y 361.868,Z 673.197,A -85,B 0,C 180,E1 -13102.982,E2 -13102.982} C_VEL
LIN {X 0,Y 361.852,Z 673.22,A -85,B 0,C 180,E1 -13106.63,E2 -13106.63} C_VEL
LIN {X 0,Y 361.869,Z 673.181,A -85,B 0,C 180,E1 -13109.671,E2 -13109.671} C_VEL
LIN {X 0,Y 361.947,Z 673.189,A -85,B 0,C 180,E1 -13113.474,E2 -13113.474} C_VEL
LIN {X 0,Y 361.883,Z 673.204,A -85,B 0,C 180,E1 -13117.144,E2 -13117.144} C_VEL
LIN {X 0,Y 361.919,Z 673.209,A -85,B 0,C 180,E1 -13120.724,E2 -13120.724} C_VEL
LIN {X 0,Y 361.938,Z 673.212,A -85,B 0,C 180,E1 -13124.226,E2 -13124.226} C_VEL
LIN {X 0,Y 361.992,Z 673.192,A -85,B 0,C 180,E1 -13126.527,E2 -13126.527} C_VEL
LIN {X 0,Y 362.028,Z 673.198,A -85,B 0,C 180,E1 -13129.938,E2 -13129.938} C_VEL
LIN {X 0,Y 362.16,Z 673.173,A -85,B 0,C 180,E1 -13133.313,E2 -13133.313} C_VEL
LIN {X 0,Y 362.274,Z 673.155,A -85,B 0,C 180,E1 -13137.776,E2 -13137.776} C_VEL
LIN {X 0,Y 362.42,Z 673.151,A -85,B 0,C 180,E1 -13140,E2 -13140} C_VEL
LIN {X 0,Y 362.274,Z 673.15,A -85,B 0,C 180,E1 -13142.223,E2 -13142.223} C_VEL
LIN {X 0,Y 362.157,Z 673.177,A -85,B 0,C 180,E1 -13146.686,E2 -13146.686} C_VEL
LIN {X 0,Y 362.024,Z 673.203,A -85,B 0,C 180,E1 -13150.062,E2 -13150.062} C_VEL
LIN {X 0,Y 361.988,Z 673.193,A -85,B 0,C 180,E1 -13153.899,E2 -13153.899} C_VEL
LIN {X 0,Y 361.959,Z 673.195,A -85,B 0,C 180,E1 -13157.939,E2 -13157.939} C_VEL
LIN {X 0,Y 361.908,Z 673.206,A -85,B 0,C 180,E1 -13161.651,E2 -13161.651} C_VEL
LIN {X 0,Y 361.921,Z 673.212,A -85,B 0,C 180,E1 -13165.29,E2 -13165.29} C_VEL
LIN {X 0,Y 361.913,Z 673.167,A -85,B 0,C 180,E1 -13167.778,E2 -13167.778} C_VEL
LIN {X 0,Y 361.838,Z 673.211,A -85,B 0,C 180,E1 -13171.286,E2 -13171.286} C_VEL
LIN {X 0,Y 361.846,Z 673.202,A -85,B 0,C 180,E1 -13174.281,E2 -13174.281} C_VEL
LIN {X 0,Y 361.857,Z 673.185,A -85,B 0,C 180,E1 -13177.224,E2 -13177.224} C_VEL
LIN {X 0,Y 361.898,Z 673.22,A -85,B 0,C 180,E1 -13180.769,E2 -13180.769} C_VEL
LIN {X 0,Y 361.903,Z 673.218,A -85,B 0,C 180,E1 -13184.354,E2 -13184.354} C_VEL
LIN {X 0,Y 361.85,Z 673.224,A -85,B 0,C 180,E1 -13187.565,E2 -13187.565} C_VEL
LIN {X 0,Y 361.868,Z 673.224,A -85,B 0,C 180,E1 -13190.973,E2 -13190.973} C_VEL
LIN {X 0,Y 361.868,Z 673.222,A -85,B 0,C 180,E1 -13194.656,E2 -13194.656} C_VEL
LIN {X 0,Y 361.832,Z 673.226,A -85,B 0,C 180,E1 -13198.371,E2 -13198.371} C_VEL
LIN {X 0,Y 361.885,Z 673.363,A -85,B 0,C 180,E1 -13199.995,E2 -13199.995} C_VEL
LIN {X 0,Y 362.216,Z 674.609,A -85,B 0,C 180,E1 -13200.633,E2 -13200.633} C_VEL
LIN {X 0,Y 363.596,Z 676.973,A -85,B 0,C 180,E1 -13201.432,E2 -13201.432} C_VEL
LIN {X 0,Y 365.775,Z 678.705,A -85,B 0,C 180,E1 -13202.54,E2 -13202.54} C_VEL
LIN {X 0,Y 367.514,Z 679.884,A -85,B 0,C 180,E1 -13203.424,E2 -13203.424} C_VEL
LIN {X 0,Y 369.12,Z 682.745,A -85,B 0,C 180,E1 -13204.408,E2 -13204.408} C_VEL
LIN {X 0,Y 371.563,Z 684.712,A -85,B 0,C 180,E1 -13205.786,E2 -13205.786} C_VEL
LIN {X 0,Y 373.135,Z 685.76,A -85,B 0,C 180,E1 -13206.701,E2 -13206.701} C_VEL
LIN {X 0,Y 374.941,Z 688.702,A -85,B 0,C 180,E1 -13207.911,E2 -13207.911} C_VEL
LIN {X 0,Y 377.178,Z 690.567,A -85,B 0,C 180,E1 -13209.367,E2 -13209.367} C_VEL
LIN {X 0,Y 379.388,Z 691.952,A -85,B 0,C 180,E1 -13210.863,E2 -13210.863} C_VEL
LIN {X 0,Y 381.206,Z 694.833,A -85,B 0,C 180,E1 -13212.33,E2 -13212.33} C_VEL
LIN {X 0,Y 383.555,Z 696.8,A -85,B 0,C 180,E1 -13214.22,E2 -13214.22} C_VEL
LIN {X 0,Y 385.859,Z 698.16,A -85,B 0,C 180,E1 -13216.304,E2 -13216.304} C_VEL
LIN {X 0,Y 387.441,Z 700.765,A -85,B 0,C 180,E1 -13218.093,E2 -13218.093} C_VEL
LIN {X 0,Y 389.003,Z 702.37,A -85,B 0,C 180,E1 -13220.09,E2 -13220.09} C_VEL
LIN {X 0,Y 390.776,Z 703.37,A -85,B 0,C 180,E1 -13222.768,E2 -13222.768} C_VEL
LIN {X 0,Y 392.01,Z 704.1,A -85,B 0,C 180,E1 -13225.484,E2 -13225.484} C_VEL
LIN {X 0,Y 392.655,Z 704.34,A -85,B 0,C 180,E1 -13227.949,E2 -13227.949} C_VEL
LIN {X 0,Y 392.856,Z 704.405,A -85,B 0,C 180,E1 -13230,E2 -13230} C_VEL
LIN {X 0,Y 392.655,Z 704.342,A -85,B 0,C 180,E1 -13232.051,E2 -13232.051} C_VEL
LIN {X 0,Y 392.01,Z 704.098,A -85,B 0,C 180,E1 -13234.515,E2 -13234.515} C_VEL
LIN {X 0,Y 390.776,Z 703.371,A -85,B 0,C 180,E1 -13237.232,E2 -13237.232} C_VEL
LIN {X 0,Y 389.094,Z 702.447,A -85,B 0,C 180,E1 -13239.788,E2 -13239.788} C_VEL
LIN {X 0,Y 387.339,Z 700.662,A -85,B 0,C 180,E1 -13242.014,E2 -13242.014} C_VEL
LIN {X 0,Y 385.578,Z 697.874,A -85,B 0,C 180,E1 -13243.975,E2 -13243.975} C_VEL
LIN {X 0,Y 382.777,Z 696.306,A -85,B 0,C 180,E1 -13246.397,E2 -13246.397} C_VEL
LIN {X 0,Y 380.67,Z 694.104,A -85,B 0,C 180,E1 -13248.109,E2 -13248.109} C_VEL
LIN {X 0,Y 378.901,Z 691.42,A -85,B 0,C 180,E1 -13249.503,E2 -13249.503} C_VEL
LIN {X 0,Y 375.918,Z 689.683,A -85,B 0,C 180,E1 -13251.459,E2 -13251.459} C_VEL
LIN {X 0,Y 373.942,Z 687.246,A -85,B 0,C 180,E1 -13252.762,E2 -13252.762} C_VEL
LIN {X 0,Y 372.81,Z 685.346,A -85,B 0,C 180,E1 -13253.508,E2 -13253.508} C_VEL
LIN {X 0,Y 369.762,Z 683.397,A -85,B 0,C 180,E1 -13255.243,E2 -13255.243} C_VEL
LIN {X 0,Y 368.027,Z 681.036,A -85,B 0,C 180,E1 -13256.241,E2 -13256.241} C_VEL
LIN {X 0,Y 367.121,Z 679.482,A -85,B 0,C 180,E1 -13256.783,E2 -13256.783} C_VEL
LIN {X 0,Y 364.002,Z 677.405,A -85,B 0,C 180,E1 -13258.362,E2 -13258.362} C_VEL
LIN {X 0,Y 362.359,Z 674.994,A -85,B 0,C 180,E1 -13259.269,E2 -13259.269} C_VEL
LIN {X 0,Y 361.985,Z 673.813,A -85,B 0,C 180,E1 -13259.675,E2 -13259.675} C_VEL
LIN {X 0,Y 361.871,Z 673.255,A -85,B 0,C 180,E1 -13260.327,E2 -13260.327} C_VEL
LIN {X 0,Y 361.848,Z 673.224,A -85,B 0,C 180,E1 -13264.28,E2 -13264.28} C_VEL
LIN {X 0,Y 361.865,Z 673.222,A -85,B 0,C 180,E1 -13267.224,E2 -13267.224} C_VEL
LIN {X 0,Y 361.866,Z 673.223,A -85,B 0,C 180,E1 -13270.762,E2 -13270.762} C_VEL
LIN {X 0,Y 361.858,Z 673.225,A -85,B 0,C 180,E1 -13274.361,E2 -13274.361} C_VEL
LIN {X 0,Y 361.876,Z 673.222,A -85,B 0,C 180,E1 -13277.559,E2 -13277.559} C_VEL
LIN {X 0,Y 361.876,Z 673.22,A -85,B 0,C 180,E1 -13279.606,E2 -13279.606} C_VEL
LIN {X 0,Y 361.195,Z 673.308,A -85,B 0,C 180,E1 -13280.534,E2 -13280.534} C_VEL
LIN {X 0,Y 358.344,Z 673.636,A -85,B 0,C 180,E1 -13282.044,E2 -13282.044} C_VEL
LIN {X 0,Y 355.933,Z 673.919,A -85,B 0,C 180,E1 -13283.266,E2 -13283.266} C_VEL
LIN {X 0,Y 354.893,Z 674.045,A -85,B 0,C 180,E1 -13284.211,E2 -13284.211} C_VEL
LIN {X 0,Y 354.805,Z 674.058,A -85,B 0,C 180,E1 -13284.531,E2 -13284.531} C_VEL
LIN {X 0,Y 354.779,Z 674.105,A -85,B 0,C 180,E1 -13287.666,E2 -13287.666} C_VEL
LIN {X 0,Y 354.86,Z 674.042,A -85,B 0,C 180,E1 -13290.621,E2 -13290.621} C_VEL
LIN {X 0,Y 354.891,Z 674.079,A -85,B 0,C 180,E1 -13294.173,E2 -13294.173} C_VEL
LIN {X 0,Y 354.844,Z 674.083,A -85,B 0,C 180,E1 -13297.895,E2 -13297.895} C_VEL
LIN {X 0,Y 354.915,Z 674.072,A -85,B 0,C 180,E1 -13301.891,E2 -13301.891} C_VEL
LIN {X 0,Y 354.933,Z 674.073,A -85,B 0,C 180,E1 -13305.982,E2 -13305.982} C_VEL
LIN {X 0,Y 354.97,Z 674.078,A -85,B 0,C 180,E1 -13309.736,E2 -13309.736} C_VEL
LIN {X 0,Y 355.121,Z 674.049,A -85,B 0,C 180,E1 -13313.181,E2 -13313.181} C_VEL
LIN {X 0,Y 355.237,Z 674.027,A -85,B 0,C 180,E1 -13317.733,E2 -13317.733} C_VEL
LIN {X 0,Y 355.39,Z 674.028,A -85,B 0,C 180,E1 -13320,E2 -13320} C_VEL
LIN {X 0,Y 355.237,Z 674.031,A -85,B 0,C 180,E1 -13322.268,E2 -13322.268} C_VEL
LIN {X 0,Y 355.124,Z 674.048,A -85,B 0,C 180,E1 -13326.82,E2 -13326.82} C_VEL
LIN {X 0,Y 354.975,Z 674.076,A -85,B 0,C 180,E1 -13330.264,E2 -13330.264} C_VEL
LIN {X 0,Y 354.935,Z 674.074,A -85,B 0,C 180,E1 -13334.02,E2 -13334.02} C_VEL
LIN {X 0,Y 354.916,Z 674.071,A -85,B 0,C 180,E1 -13338.109,E2 -13338.109} C_VEL
LIN {X 0,Y 354.83,Z 674.082,A -85,B 0,C 180,E1 -13342.106,E2 -13342.106} C_VEL
LIN {X 0,Y 354.892,Z 674.081,A -85,B 0,C 180,E1 -13345.828,E2 -13345.828} C_VEL
LIN {X 0,Y 354.848,Z 674.043,A -85,B 0,C 180,E1 -13349.679,E2 -13349.679} C_VEL
LIN {X 0,Y 354.8,Z 674.091,A -85,B 0,C 180,E1 -13353.703,E2 -13353.703} C_VEL
LIN {X 0,Y 354.795,Z 674.07,A -85,B 0,C 180,E1 -13356.46,E2 -13356.46} C_VEL
LIN {X 0,Y 354.819,Z 674.091,A -85,B 0,C 180,E1 -13359.424,E2 -13359.424} C_VEL
LIN {X 0,Y 354.831,Z 674.089,A -85,B 0,C 180,E1 -13362.876,E2 -13362.876} C_VEL
LIN {X 0,Y 354.832,Z 674.146,A -85,B 0,C 180,E1 -13365.482,E2 -13365.482} C_VEL
LIN {X 0,Y 355.587,Z 676.925,A -85,B 0,C 180,E1 -13366.438,E2 -13366.438} C_VEL
LIN {X 0,Y 358.861,Z 688.117,A -85,B 0,C 180,E1 -13369.799,E2 -13369.799} C_VEL
LIN {X 0,Y 359.338,Z 689.607,A -85,B 0,C 180,E1 -13370.09,E2 -13370.09} C_VEL
LIN {X 0,Y 369.4,Z 708.292,A -85,B 0,C 180,E1 -13371.84,E2 -13371.84} C_VEL
LIN {X 0,Y 377.64,Z 725.211,A -85,B 0,C 180,E1 -13373.202,E2 -13373.202} C_VEL
LIN {X 0,Y 379.632,Z 729.844,A -85,B 0,C 180,E1 -13373.532,E2 -13373.532} C_VEL
LIN {X 0,Y 382.78,Z 744.799,A -85,B 0,C 180,E1 -13374.215,E2 -13374.215} C_VEL
LIN {X 0,Y 378.198,Z 892.796,A -85,B 0,C 180,E1 -13377.09,E2 -13377.09} C_VEL
LIN {X 0,Y 377.447,Z 904.443,A -85,B 0,C 180,E1 -13377.398,E2 -13377.398} C_VEL
LIN {X 0,Y 376.215,Z 917.776,A -85,B 0,C 180,E1 -13377.873,E2 -13377.873} C_VEL
LIN {X 0,Y 374.895,Z 930.897,A -85,B 0,C 180,E1 -13378.497,E2 -13378.497} C_VEL
LIN {X 0,Y 373.536,Z 942.284,A -85,B 0,C 180,E1 -13379.157,E2 -13379.157} C_VEL
LIN {X 0,Y 371.664,Z 955.52,A -85,B 0,C 180,E1 -13380.084,E2 -13380.084} C_VEL
LIN {X 0,Y 369.721,Z 968.207,A -85,B 0,C 180,E1 -13381.156,E2 -13381.156} C_VEL
LIN {X 0,Y 367.797,Z 979.256,A -85,B 0,C 180,E1 -13382.241,E2 -13382.241} C_VEL
LIN {X 0,Y 365.869,Z 990.058,A -85,B 0,C 180,E1 -13383.474,E2 -13383.474} C_VEL
LIN {X 0,Y 363.846,Z 1000.557,A -85,B 0,C 180,E1 -13384.853,E2 -13384.853} C_VEL
LIN {X 0,Y 362.079,Z 1009.829,A -85,B 0,C 180,E1 -13386.25,E2 -13386.25} C_VEL
LIN {X 0,Y 360.21,Z 1019.564,A -85,B 0,C 180,E1 -13387.94,E2 -13387.94} C_VEL
LIN {X 0,Y 358.55,Z 1028.089,A -85,B 0,C 180,E1 -13389.64,E2 -13389.64} C_VEL
LIN {X 0,Y 357.066,Z 1036.694,A -85,B 0,C 180,E1 -13391.644,E2 -13391.644} C_VEL
LIN {X 0,Y 355.882,Z 1043.123,A -85,B 0,C 180,E1 -13393.361,E2 -13393.361} C_VEL
LIN {X 0,Y 354.794,Z 1050.388,A -85,B 0,C 180,E1 -13395.665,E2 -13395.665} C_VEL
LIN {X 0,Y 354.223,Z 1055.039,A -85,B 0,C 180,E1 -13397.394,E2 -13397.394} C_VEL
LIN {X 0,Y 353.619,Z 1060.135,A -85,B 0,C 180,E1 -13399.696,E2 -13399.696} C_VEL
LIN {X 0,Y 353.373,Z 1064.134,A -85,B 0,C 180,E1 -13401.998,E2 -13401.998} C_VEL
LIN {X 0,Y 353.26,Z 1067.088,A -85,B 0,C 180,E1 -13404.291,E2 -13404.291} C_VEL
LIN {X 0,Y 353.223,Z 1068.272,A -85,B 0,C 180,E1 -13405.435,E2 -13405.435} C_VEL
LIN {X 0,Y 353.159,Z 1069.737,A -85,B 0,C 180,E1 -13407.719,E2 -13407.719} C_VEL
LIN {X 0,Y 353.259,Z 1070.226,A -85,B 0,C 180,E1 -13410,E2 -13410} C_VEL
LIN {X 0,Y 353.159,Z 1069.737,A -85,B 0,C 180,E1 -13412.281,E2 -13412.281} C_VEL
LIN {X 0,Y 353.223,Z 1068.272,A -85,B 0,C 180,E1 -13414.565,E2 -13414.565} C_VEL
LIN {X 0,Y 353.299,Z 1065.807,A -85,B 0,C 180,E1 -13416.855,E2 -13416.855} C_VEL
LIN {X 0,Y 353.543,Z 1061.223,A -85,B 0,C 180,E1 -13419.728,E2 -13419.728} C_VEL
LIN {X 0,Y 353.908,Z 1057.736,A -85,B 0,C 180,E1 -13421.454,E2 -13421.454} C_VEL
LIN {X 0,Y 354.632,Z 1051.846,A -85,B 0,C 180,E1 -13423.816,E2 -13423.816} C_VEL
LIN {X 0,Y 355.288,Z 1046.947,A -85,B 0,C 180,E1 -13425.488,E2 -13425.488} C_VEL
LIN {X 0,Y 356.706,Z 1038.918,A -85,B 0,C 180,E1 -13427.781,E2 -13427.781} C_VEL
LIN {X 0,Y 357.901,Z 1031.873,A -85,B 0,C 180,E1 -13429.514,E2 -13429.514} C_VEL
LIN {X 0,Y 359.351,Z 1023.96,A -85,B 0,C 180,E1 -13431.211,E2 -13431.211} C_VEL
LIN {X 0,Y 361.089,Z 1014.846,A -85,B 0,C 180,E1 -13432.908,E2 -13432.908} C_VEL
LIN {X 0,Y 363.054,Z 1004.841,A -85,B 0,C 180,E1 -13434.519,E2 -13434.519} C_VEL
LIN {X 0,Y 365.037,Z 994.41,A -85,B 0,C 180,E1 -13435.976,E2 -13435.976} C_VEL
LIN {X 0,Y 367.05,Z 982.994,A -85,B 0,C 180,E1 -13437.356,E2 -13437.356} C_VEL
LIN {X 0,Y 368.958,Z 972.574,A -85,B 0,C 180,E1 -13438.437,E2 -13438.437} C_VEL
LIN {X 0,Y 370.932,Z 960.548,A -85,B 0,C 180,E1 -13439.512,E2 -13439.512} C_VEL
LIN {X 0,Y 372.683,Z 948.226,A -85,B 0,C 180,E1 -13440.45,E2 -13440.45} C_VEL
LIN {X 0,Y 374.363,Z 935.684,A -85,B 0,C 180,E1 -13441.238,E2 -13441.238} C_VEL
LIN {X 0,Y 375.777,Z 922.253,A -85,B 0,C 180,E1 -13441.932,E2 -13441.932} C_VEL
LIN {X 0,Y 377.031,Z 909.337,A -85,B 0,C 180,E1 -13442.444,E2 -13442.444} C_VEL
LIN {X 0,Y 378.113,Z 895.393,A -85,B 0,C 180,E1 -13442.845,E2 -13442.845} C_VEL
LIN {X 0,Y 379.108,Z 863.628,A -85,B 0,C 180,E1 -13443.502,E2 -13443.502} C_VEL
LIN {X 0,Y 382.781,Z 744.478,A -85,B 0,C 180,E1 -13445.792,E2 -13445.792} C_VEL
LIN {X 0,Y 379.367,Z 729.117,A -85,B 0,C 180,E1 -13446.514,E2 -13446.514} C_VEL
LIN {X 0,Y 371.089,Z 711.443,A -85,B 0,C 180,E1 -13447.882,E2 -13447.882} C_VEL
LIN {X 0,Y 361.076,Z 692.808,A -85,B 0,C 180,E1 -13449.587,E2 -13449.587} C_VEL
LIN {X 0,Y 359.105,Z 688.928,A -85,B 0,C 180,E1 -13450.002,E2 -13450.002} C_VEL
LIN {X 0,Y 356.094,Z 678.416,A -85,B 0,C 180,E1 -13453.093,E2 -13453.093} C_VEL
LIN {X 0,Y 354.848,Z 674.368,A -85,B 0,C 180,E1 -13454.388,E2 -13454.388} C_VEL
LIN {X 0,Y 354.83,Z 674.077,A -85,B 0,C 180,E1 -13454.945,E2 -13454.945} C_VEL
LIN {X 0,Y 354.833,Z 674.069,A -85,B 0,C 180,E1 -13458.818,E2 -13458.818} C_VEL
LIN {X 0,Y 354.808,Z 674.087,A -85,B 0,C 180,E1 -13462.401,E2 -13462.401} C_VEL
LIN {X 0,Y 354.806,Z 674.069,A -85,B 0,C 180,E1 -13464.94,E2 -13464.94} C_VEL
LIN {X 0,Y 354.787,Z 674.095,A -85,B 0,C 180,E1 -13468.404,E2 -13468.404} C_VEL
LIN {X 0,Y 354.846,Z 674.039,A -85,B 0,C 180,E1 -13471.619,E2 -13471.619} C_VEL
LIN {X 0,Y 354.892,Z 674.081,A -85,B 0,C 180,E1 -13474.172,E2 -13474.172} C_VEL
LIN {X 0,Y 354.83,Z 674.082,A -85,B 0,C 180,E1 -13477.894,E2 -13477.894} C_VEL
LIN {X 0,Y 354.916,Z 674.072,A -85,B 0,C 180,E1 -13481.891,E2 -13481.891} C_VEL
LIN {X 0,Y 354.935,Z 674.076,A -85,B 0,C 180,E1 -13485.98,E2 -13485.98} C_VEL
LIN {X 0,Y 354.975,Z 674.077,A -85,B 0,C 180,E1 -13489.736,E2 -13489.736} C_VEL
LIN {X 0,Y 355.124,Z 674.047,A -85,B 0,C 180,E1 -13493.18,E2 -13493.18} C_VEL
LIN {X 0,Y 355.237,Z 674.03,A -85,B 0,C 180,E1 -13497.732,E2 -13497.732} C_VEL
LIN {X 0,Y 355.39,Z 674.026,A -85,B 0,C 180,E1 -13500,E2 -13500} C_VEL
LIN {X 0,Y 355.237,Z 674.026,A -85,B 0,C 180,E1 -13502.267,E2 -13502.267} C_VEL
LIN {X 0,Y 355.121,Z 674.051,A -85,B 0,C 180,E1 -13506.819,E2 -13506.819} C_VEL
LIN {X 0,Y 354.97,Z 674.08,A -85,B 0,C 180,E1 -13510.264,E2 -13510.264} C_VEL
LIN {X 0,Y 354.933,Z 674.074,A -85,B 0,C 180,E1 -13514.018,E2 -13514.018} C_VEL
LIN {X 0,Y 354.915,Z 674.072,A -85,B 0,C 180,E1 -13518.109,E2 -13518.109} C_VEL
LIN {X 0,Y 354.844,Z 674.083,A -85,B 0,C 180,E1 -13522.105,E2 -13522.105} C_VEL
LIN {X 0,Y 354.891,Z 674.079,A -85,B 0,C 180,E1 -13525.827,E2 -13525.827} C_VEL
LIN {X 0,Y 354.846,Z 674.047,A -85,B 0,C 180,E1 -13529.679,E2 -13529.679} C_VEL
LIN {X 0,Y 354.798,Z 674.093,A -85,B 0,C 180,E1 -13533.702,E2 -13533.702} C_VEL
LIN {X 0,Y 354.79,Z 674.057,A -85,B 0,C 180,E1 -13536.46,E2 -13536.46} C_VEL
LIN {X 0,Y 354.816,Z 674.102,A -85,B 0,C 180,E1 -13539.424,E2 -13539.424} C_VEL
LIN {X 0,Y 354.827,Z 674.101,A -85,B 0,C 180,E1 -13542.876,E2 -13542.876} C_VEL
LIN {X 0,Y 354.797,Z 674.103,A -85,B 0,C 180,E1 -13546.11,E2 -13546.11} C_VEL
LIN {X 0,Y 354.818,Z 674.101,A -85,B 0,C 180,E1 -13549.185,E2 -13549.185} C_VEL
LIN {X 0,Y 354.803,Z 674.103,A -85,B 0,C 180,E1 -13552.403,E2 -13552.403} C_VEL
LIN {X 0,Y 354.806,Z 674.103,A -85,B 0,C 180,E1 -13554.941,E2 -13554.941} C_VEL
LIN {X 0,Y 354.848,Z 674.365,A -85,B 0,C 180,E1 -13557.169,E2 -13557.169} C_VEL
LIN {X 0,Y 355.129,Z 675.607,A -85,B 0,C 180,E1 -13557.679,E2 -13557.679} C_VEL
LIN {X 0,Y 356.344,Z 677.733,A -85,B 0,C 180,E1 -13558.318,E2 -13558.318} C_VEL
LIN {X 0,Y 358.892,Z 679.698,A -85,B 0,C 180,E1 -13559.499,E2 -13559.499} C_VEL
LIN {X 0,Y 360.197,Z 680.677,A -85,B 0,C 180,E1 -13560.131,E2 -13560.131} C_VEL
LIN {X 0,Y 361.925,Z 683.464,A -85,B 0,C 180,E1 -13561.053,E2 -13561.053} C_VEL
LIN {X 0,Y 364.331,Z 685.498,A -85,B 0,C 180,E1 -13562.266,E2 -13562.266} C_VEL
LIN {X 0,Y 365.931,Z 686.485,A -85,B 0,C 180,E1 -13563.087,E2 -13563.087} C_VEL
LIN {X 0,Y 367.572,Z 689.322,A -85,B 0,C 180,E1 -13564.064,E2 -13564.064} C_VEL
LIN {X 0,Y 369.745,Z 691.273,A -85,B 0,C 180,E1 -13565.282,E2 -13565.282} C_VEL
LIN {X 0,Y 371.773,Z 692.519,A -85,B 0,C 180,E1 -13566.422,E2 -13566.422} C_VEL
LIN {X 0,Y 373.612,Z 695.419,A -85,B 0,C 180,E1 -13567.628,E2 -13567.628} C_VEL
LIN {X 0,Y 376.035,Z 697.501,A -85,B 0,C 180,E1 -13569.201,E2 -13569.201} C_VEL
LIN {X 0,Y 378.222,Z 698.881,A -85,B 0,C 180,E1 -13570.671,E2 -13570.671} C_VEL
LIN {X 0,Y 380.059,Z 701.716,A -85,B 0,C 180,E1 -13572.134,E2 -13572.134} C_VEL
LIN {X 0,Y 382.392,Z 703.713,A -85,B 0,C 180,E1 -13573.998,E2 -13573.998} C_VEL
LIN {X 0,Y 384.802,Z 705.084,A -85,B 0,C 180,E1 -13576.131,E2 -13576.131} C_VEL
LIN {X 0,Y 386.429,Z 707.731,A -85,B 0,C 180,E1 -13577.958,E2 -13577.958} C_VEL
LIN {X 0,Y 388.115,Z 709.415,A -85,B 0,C 180,E1 -13580.068,E2 -13580.068} C_VEL
LIN {X 0,Y 389.898,Z 710.415,A -85,B 0,C 180,E1 -13582.752,E2 -13582.752} C_VEL
LIN {X 0,Y 391.14,Z 711.147,A -85,B 0,C 180,E1 -13585.474,E2 -13585.474} C_VEL
LIN {X 0,Y 391.79,Z 711.387,A -85,B 0,C 180,E1 -13587.944,E2 -13587.944} C_VEL
LIN {X 0,Y 391.991,Z 711.452,A -85,B 0,C 180,E1 -13590,E2 -13590} C_VEL
LIN {X 0,Y 391.79,Z 711.39,A -85,B 0,C 180,E1 -13592.056,E2 -13592.056} C_VEL
LIN {X 0,Y 391.14,Z 711.144,A -85,B 0,C 180,E1 -13594.525,E2 -13594.525} C_VEL
LIN {X 0,Y 389.899,Z 710.416,A -85,B 0,C 180,E1 -13597.248,E2 -13597.248} C_VEL
LIN {X 0,Y 388.206,Z 709.491,A -85,B 0,C 180,E1 -13599.811,E2 -13599.811} C_VEL
LIN {X 0,Y 386.43,Z 707.724,A -85,B 0,C 180,E1 -13602.042,E2 -13602.042} C_VEL
LIN {X 0,Y 384.525,Z 704.811,A -85,B 0,C 180,E1 -13604.149,E2 -13604.149} C_VEL
LIN {X 0,Y 381.665,Z 703.207,A -85,B 0,C 180,E1 -13606.583,E2 -13606.583} C_VEL
LIN {X 0,Y 379.39,Z 700.8,A -85,B 0,C 180,E1 -13608.425,E2 -13608.425} C_VEL
LIN {X 0,Y 377.934,Z 698.493,A -85,B 0,C 180,E1 -13609.555,E2 -13609.555} C_VEL
LIN {X 0,Y 374.562,Z 696.443,A -85,B 0,C 180,E1 -13611.74,E2 -13611.74} C_VEL
LIN {X 0,Y 372.474,Z 693.83,A -85,B 0,C 180,E1 -13613.098,E2 -13613.098} C_VEL
LIN {X 0,Y 371.567,Z 692.204,A -85,B 0,C 180,E1 -13613.716,E2 -13613.716} C_VEL
LIN {X 0,Y 368.524,Z 690.314,A -85,B 0,C 180,E1 -13615.409,E2 -13615.409} C_VEL
LIN {X 0,Y 366.655,Z 687.916,A -85,B 0,C 180,E1 -13616.49,E2 -13616.49} C_VEL
LIN {X 0,Y 365.533,Z 686.101,A -85,B 0,C 180,E1 -13617.123,E2 -13617.123} C_VEL
LIN {X 0,Y 362.852,Z 684.424,A -85,B 0,C 180,E1 -13618.468,E2 -13618.468} C_VEL
LIN {X 0,Y 360.82,Z 681.84,A -85,B 0,C 180,E1 -13619.537,E2 -13619.537} C_VEL
LIN {X 0,Y 359.794,Z 680.199,A -85,B 0,C 180,E1 -13620.072,E2 -13620.072} C_VEL
LIN {X 0,Y 356.851,Z 678.281,A -85,B 0,C 180,E1 -13621.435,E2 -13621.435} C_VEL
LIN {X 0,Y 355.27,Z 675.978,A -85,B 0,C 180,E1 -13622.236,E2 -13622.236} C_VEL
LIN {X 0,Y 354.887,Z 674.626,A -85,B 0,C 180,E1 -13622.658,E2 -13622.658} C_VEL
LIN {X 0,Y 354.81,Z 674.188,A -85,B 0,C 180,E1 -13623.004,E2 -13623.004} C_VEL
LIN {X 0,Y 354.796,Z 674.105,A -85,B 0,C 180,E1 -13626.459,E2 -13626.459} C_VEL
LIN {X 0,Y 354.818,Z 674.1,A -85,B 0,C 180,E1 -13629.423,E2 -13629.423} C_VEL
LIN {X 0,Y 354.8,Z 674.102,A -85,B 0,C 180,E1 -13632.87,E2 -13632.87} C_VEL
LIN {X 0,Y 354.844,Z 674.098,A -85,B 0,C 180,E1 -13636.116,E2 -13636.116} C_VEL
LIN {X 0,Y 354.818,Z 674.099,A -85,B 0,C 180,E1 -13639.596,E2 -13639.596} C_VEL
LIN {X 0,Y 354.79,Z 674.057,A -85,B 0,C 180,E1 -13643.54,E2 -13643.54} C_VEL
LIN {X 0,Y 354.805,Z 674.058,A -85,B 0,C 180,E1 -13644.531,E2 -13644.531} C_VEL
LIN {X 0,Y 354.115,Z 674.16,A -85,B 0,C 180,E1 -13645.478,E2 -13645.478} C_VEL
LIN {X 0,Y 351.219,Z 674.548,A -85,B 0,C 180,E1 -13647.017,E2 -13647.017} C_VEL
LIN {X 0,Y 348.803,Z 674.844,A -85,B 0,C 180,E1 -13648.263,E2 -13648.263} C_VEL
LIN {X 0,Y 347.807,Z 674.944,A -85,B 0,C 180,E1 -13649.228,E2 -13649.228} C_VEL
LIN {X 0,Y 347.748,Z 674.942,A -85,B 0,C 180,E1 -13649.555,E2 -13649.555} C_VEL
LIN {X 0,Y 347.844,Z 674.925,A -85,B 0,C 180,E1 -13652.744,E2 -13652.744} C_VEL
LIN {X 0,Y 347.79,Z 674.971,A -85,B 0,C 180,E1 -13656.163,E2 -13656.163} C_VEL
LIN {X 0,Y 347.827,Z 674.973,A -85,B 0,C 180,E1 -13659.911,E2 -13659.911} C_VEL
LIN {X 0,Y 347.858,Z 674.949,A -85,B 0,C 180,E1 -13662.359,E2 -13662.359} C_VEL
LIN {X 0,Y 347.889,Z 674.95,A -85,B 0,C 180,E1 -13665.971,E2 -13665.971} C_VEL
LIN {X 0,Y 347.921,Z 674.955,A -85,B 0,C 180,E1 -13669.526,E2 -13669.526} C_VEL
LIN {X 0,Y 348.086,Z 674.923,A -85,B 0,C 180,E1 -13673.042,E2 -13673.042} C_VEL
LIN {X 0,Y 348.2,Z 674.903,A -85,B 0,C 180,E1 -13677.687,E2 -13677.687} C_VEL
LIN {X 0,Y 348.359,Z 674.904,A -85,B 0,C 180,E1 -13680,E2 -13680} C_VEL
LIN {X 0,Y 348.2,Z 674.907,A -85,B 0,C 180,E1 -13682.314,E2 -13682.314} C_VEL
LIN {X 0,Y 348.089,Z 674.921,A -85,B 0,C 180,E1 -13686.958,E2 -13686.958} C_VEL
LIN {X 0,Y 347.925,Z 674.955,A -85,B 0,C 180,E1 -13690.475,E2 -13690.475} C_VEL
LIN {X 0,Y 347.891,Z 674.952,A -85,B 0,C 180,E1 -13694.15,E2 -13694.15} C_VEL
LIN {X 0,Y 347.884,Z 674.948,A -85,B 0,C 180,E1 -13698.291,E2 -13698.291} C_VEL
LIN {X 0,Y 347.788,Z 674.963,A -85,B 0,C 180,E1 -13701.638,E2 -13701.638} C_VEL
LIN {X 0,Y 347.806,Z 674.974,A -85,B 0,C 180,E1 -13705.109,E2 -13705.109} C_VEL
LIN {X 0,Y 347.805,Z 674.921,A -85,B 0,C 180,E1 -13707.694,E2 -13707.694} C_VEL
LIN {X 0,Y 347.758,Z 674.935,A -85,B 0,C 180,E1 -13710.347,E2 -13710.347} C_VEL
LIN {X 0,Y 347.738,Z 674.956,A -85,B 0,C 180,E1 -13714.465,E2 -13714.465} C_VEL
LIN {X 0,Y 347.774,Z 674.973,A -85,B 0,C 180,E1 -13717.991,E2 -13717.991} C_VEL
LIN {X 0,Y 347.778,Z 674.95,A -85,B 0,C 180,E1 -13721.826,E2 -13721.826} C_VEL
LIN {X 0,Y 347.827,Z 675.105,A -85,B 0,C 180,E1 -13724.744,E2 -13724.744} C_VEL
LIN {X 0,Y 350.653,Z 684.817,A -85,B 0,C 180,E1 -13727.866,E2 -13727.866} C_VEL
LIN {X 0,Y 351.867,Z 688.956,A -85,B 0,C 180,E1 -13729.044,E2 -13729.044} C_VEL
LIN {X 0,Y 360.206,Z 704.117,A -85,B 0,C 180,E1 -13730.585,E2 -13730.585} C_VEL
LIN {X 0,Y 368.583,Z 720.484,A -85,B 0,C 180,E1 -13732.036,E2 -13732.036} C_VEL
LIN {X 0,Y 374.334,Z 733.228,A -85,B 0,C 180,E1 -13733.014,E2 -13733.014} C_VEL
LIN {X 0,Y 376.982,Z 746.234,A -85,B 0,C 180,E1 -13733.616,E2 -13733.616} C_VEL
LIN {X 0,Y 372.265,Z 891.922,A -85,B 0,C 180,E1 -13736.478,E2 -13736.478} C_VEL
LIN {X 0,Y 371.486,Z 904.237,A -85,B 0,C 180,E1 -13736.808,E2 -13736.808} C_VEL
LIN {X 0,Y 370.224,Z 917.571,A -85,B 0,C 180,E1 -13737.288,E2 -13737.288} C_VEL
LIN {X 0,Y 368.822,Z 930.69,A -85,B 0,C 180,E1 -13737.917,E2 -13737.917} C_VEL
LIN {X 0,Y 367.437,Z 942.078,A -85,B 0,C 180,E1 -13738.587,E2 -13738.587} C_VEL
LIN {X 0,Y 365.47,Z 955.313,A -85,B 0,C 180,E1 -13739.524,E2 -13739.524} C_VEL
LIN {X 0,Y 363.512,Z 967.702,A -85,B 0,C 180,E1 -13740.583,E2 -13740.583} C_VEL
LIN {X 0,Y 361.45,Z 979.048,A -85,B 0,C 180,E1 -13741.71,E2 -13741.71} C_VEL
LIN {X 0,Y 359.456,Z 989.85,A -85,B 0,C 180,E1 -13742.963,E2 -13742.963} C_VEL
LIN {X 0,Y 357.364,Z 1000.349,A -85,B 0,C 180,E1 -13744.364,E2 -13744.364} C_VEL
LIN {X 0,Y 355.512,Z 1009.621,A -85,B 0,C 180,E1 -13745.783,E2 -13745.783} C_VEL
LIN {X 0,Y 353.543,Z 1019.356,A -85,B 0,C 180,E1 -13747.502,E2 -13747.502} C_VEL
LIN {X 0,Y 351.789,Z 1027.88,A -85,B 0,C 180,E1 -13749.231,E2 -13749.231} C_VEL
LIN {X 0,Y 350.2,Z 1036.484,A -85,B 0,C 180,E1 -13751.271,E2 -13751.271} C_VEL
LIN {X 0,Y 348.99,Z 1042.915,A -85,B 0,C 180,E1 -13753.023,E2 -13753.023} C_VEL
LIN {X 0,Y 347.831,Z 1050.179,A -85,B 0,C 180,E1 -13755.371,E2 -13755.371} C_VEL
LIN {X 0,Y 347.224,Z 1054.832,A -85,B 0,C 180,E1 -13757.136,E2 -13757.136} C_VEL
LIN {X 0,Y 346.564,Z 1059.927,A -85,B 0,C 180,E1 -13759.484,E2 -13759.484} C_VEL
LIN {X 0,Y 346.282,Z 1063.926,A -85,B 0,C 180,E1 -13761.833,E2 -13761.833} C_VEL
LIN {X 0,Y 346.179,Z 1066.882,A -85,B 0,C 180,E1 -13764.174,E2 -13764.174} C_VEL
LIN {X 0,Y 346.123,Z 1068.066,A -85,B 0,C 180,E1 -13765.341,E2 -13765.341} C_VEL
LIN {X 0,Y 346.07,Z 1069.532,A -85,B 0,C 180,E1 -13767.672,E2 -13767.672} C_VEL
LIN {X 0,Y 346.162,Z 1070.021,A -85,B 0,C 180,E1 -13770,E2 -13770} C_VEL
LIN {X 0,Y 346.07,Z 1069.532,A -85,B 0,C 180,E1 -13772.328,E2 -13772.328} C_VEL
LIN {X 0,Y 346.123,Z 1068.066,A -85,B 0,C 180,E1 -13774.659,E2 -13774.659} C_VEL
LIN {X 0,Y 346.217,Z 1065.6,A -85,B 0,C 180,E1 -13776.996,E2 -13776.996} C_VEL
LIN {X 0,Y 346.489,Z 1061.016,A -85,B 0,C 180,E1 -13779.928,E2 -13779.928} C_VEL
LIN {X 0,Y 346.878,Z 1057.528,A -85,B 0,C 180,E1 -13781.689,E2 -13781.689} C_VEL
LIN {X 0,Y 347.616,Z 1051.801,A -85,B 0,C 180,E1 -13784.04,E2 -13784.04} C_VEL
LIN {X 0,Y 348.36,Z 1046.739,A -85,B 0,C 180,E1 -13785.804,E2 -13785.804} C_VEL
LIN {X 0,Y 349.841,Z 1038.709,A -85,B 0,C 180,E1 -13788.142,E2 -13788.142} C_VEL
LIN {X 0,Y 351.091,Z 1031.722,A -85,B 0,C 180,E1 -13789.895,E2 -13789.895} C_VEL
LIN {X 0,Y 352.644,Z 1023.752,A -85,B 0,C 180,E1 -13791.634,E2 -13791.634} C_VEL
LIN {X 0,Y 354.494,Z 1014.638,A -85,B 0,C 180,E1 -13793.359,E2 -13793.359} C_VEL
LIN {X 0,Y 356.366,Z 1005.419,A -85,B 0,C 180,E1 -13794.882,E2 -13794.882} C_VEL
LIN {X 0,Y 358.372,Z 995.29,A -85,B 0,C 180,E1 -13796.339,E2 -13796.339} C_VEL
LIN {X 0,Y 360.463,Z 984.034,A -85,B 0,C 180,E1 -13797.741,E2 -13797.741} C_VEL
LIN {X 0,Y 362.675,Z 972.367,A -85,B 0,C 180,E1 -13798.976,E2 -13798.976} C_VEL
LIN {X 0,Y 364.692,Z 960.34,A -85,B 0,C 180,E1 -13800.068,E2 -13800.068} C_VEL
LIN {X 0,Y 366.546,Z 948.02,A -85,B 0,C 180,E1 -13801.016,E2 -13801.016} C_VEL
LIN {X 0,Y 368.282,Z 935.477,A -85,B 0,C 180,E1 -13801.814,E2 -13801.814} C_VEL
LIN {X 0,Y 369.766,Z 922.048,A -85,B 0,C 180,E1 -13802.515,E2 -13802.515} C_VEL
LIN {X 0,Y 371.054,Z 909.132,A -85,B 0,C 180,E1 -13803.033,E2 -13803.033} C_VEL
LIN {X 0,Y 372.148,Z 895.772,A -85,B 0,C 180,E1 -13803.423,E2 -13803.423} C_VEL
LIN {X 0,Y 373.079,Z 867.805,A -85,B 0,C 180,E1 -13804.018,E2 -13804.018} C_VEL
LIN {X 0,Y 377.001,Z 746.251,A -85,B 0,C 180,E1 -13806.382,E2 -13806.382} C_VEL
LIN {X 0,Y 374.066,Z 732.347,A -85,B 0,C 180,E1 -13807.037,E2 -13807.037} C_VEL
LIN {X 0,Y 366.023,Z 715.179,A -85,B 0,C 180,E1 -13808.405,E2 -13808.405} C_VEL
LIN {X 0,Y 356.27,Z 696.896,A -85,B 0,C 180,E1 -13810.119,E2 -13810.119} C_VEL
LIN {X 0,Y 351.81,Z 688.717,A -85,B 0,C 180,E1 -13810.989,E2 -13810.989} C_VEL
LIN {X 0,Y 348.602,Z 677.939,A -85,B 0,C 180,E1 -13814.3,E2 -13814.3} C_VEL
LIN {X 0,Y 347.833,Z 675.011,A -85,B 0,C 180,E1 -13815.321,E2 -13815.321} C_VEL
LIN {X 0,Y 347.779,Z 674.948,A -85,B 0,C 180,E1 -13818.39,E2 -13818.39} C_VEL
LIN {X 0,Y 347.774,Z 674.973,A -85,B 0,C 180,E1 -13822.009,E2 -13822.009} C_VEL
LIN {X 0,Y 347.738,Z 674.956,A -85,B 0,C 180,E1 -13825.535,E2 -13825.535} C_VEL
LIN {X 0,Y 347.758,Z 674.935,A -85,B 0,C 180,E1 -13829.653,E2 -13829.653} C_VEL
LIN {X 0,Y 347.846,Z 674.923,A -85,B 0,C 180,E1 -13832.744,E2 -13832.744} C_VEL
LIN {X 0,Y 347.781,Z 674.971,A -85,B 0,C 180,E1 -13836.161,E2 -13836.161} C_VEL
LIN {X 0,Y 347.819,Z 674.972,A -85,B 0,C 180,E1 -13839.91,E2 -13839.91} C_VEL
LIN {X 0,Y 347.859,Z 674.951,A -85,B 0,C 180,E1 -13842.359,E2 -13842.359} C_VEL
LIN {X 0,Y 347.89,Z 674.953,A -85,B 0,C 180,E1 -13845.97,E2 -13845.97} C_VEL
LIN {X 0,Y 347.925,Z 674.956,A -85,B 0,C 180,E1 -13849.525,E2 -13849.525} C_VEL
LIN {X 0,Y 348.089,Z 674.921,A -85,B 0,C 180,E1 -13853.042,E2 -13853.042} C_VEL
LIN {X 0,Y 348.2,Z 674.906,A -85,B 0,C 180,E1 -13857.686,E2 -13857.686} C_VEL
LIN {X 0,Y 348.359,Z 674.902,A -85,B 0,C 180,E1 -13860,E2 -13860} C_VEL
LIN {X 0,Y 348.2,Z 674.902,A -85,B 0,C 180,E1 -13862.313,E2 -13862.313} C_VEL
LIN {X 0,Y 348.086,Z 674.925,A -85,B 0,C 180,E1 -13866.958,E2 -13866.958} C_VEL
LIN {X 0,Y 347.921,Z 674.957,A -85,B 0,C 180,E1 -13870.474,E2 -13870.474} C_VEL
LIN {X 0,Y 347.89,Z 674.952,A -85,B 0,C 180,E1 -13874.15,E2 -13874.15} C_VEL
LIN {X 0,Y 347.883,Z 674.949,A -85,B 0,C 180,E1 -13878.291,E2 -13878.291} C_VEL
LIN {X 0,Y 347.807,Z 674.961,A -85,B 0,C 180,E1 -13881.646,E2 -13881.646} C_VEL
LIN {X 0,Y 347.809,Z 674.971,A -85,B 0,C 180,E1 -13885.108,E2 -13885.108} C_VEL
LIN {X 0,Y 347.803,Z 674.923,A -85,B 0,C 180,E1 -13887.694,E2 -13887.694} C_VEL
LIN {X 0,Y 347.756,Z 674.939,A -85,B 0,C 180,E1 -13890.347,E2 -13890.347} C_VEL
LIN {X 0,Y 347.736,Z 674.952,A -85,B 0,C 180,E1 -13894.464,E2 -13894.464} C_VEL
LIN {X 0,Y 347.768,Z 674.952,A -85,B 0,C 180,E1 -13897.989,E2 -13897.989} C_VEL
LIN {X 0,Y 347.777,Z 674.978,A -85,B 0,C 180,E1 -13901.609,E2 -13901.609} C_VEL
LIN {X 0,Y 347.791,Z 674.977,A -85,B 0,C 180,E1 -13905.012,E2 -13905.012} C_VEL
LIN {X 0,Y 347.761,Z 674.979,A -85,B 0,C 180,E1 -13908.394,E2 -13908.394} C_VEL
LIN {X 0,Y 347.77,Z 674.979,A -85,B 0,C 180,E1 -13912.011,E2 -13912.011} C_VEL
LIN {X 0,Y 347.799,Z 675.123,A -85,B 0,C 180,E1 -13914.366,E2 -13914.366} C_VEL
LIN {X 0,Y 348.098,Z 676.361,A -85,B 0,C 180,E1 -13914.925,E2 -13914.925} C_VEL
LIN {X 0,Y 349.284,Z 678.575,A -85,B 0,C 180,E1 -13915.52,E2 -13915.52} C_VEL
LIN {X 0,Y 351.769,Z 680.556,A -85,B 0,C 180,E1 -13916.591,E2 -13916.591} C_VEL
LIN {X 0,Y 352.973,Z 681.507,A -85,B 0,C 180,E1 -13917.142,E2 -13917.142} C_VEL
LIN {X 0,Y 354.649,Z 684.253,A -85,B 0,C 180,E1 -13917.958,E2 -13917.958} C_VEL
LIN {X 0,Y 357.133,Z 686.344,A -85,B 0,C 180,E1 -13919.123,E2 -13919.123} C_VEL
LIN {X 0,Y 358.474,Z 687.178,A -85,B 0,C 180,E1 -13919.748,E2 -13919.748} C_VEL
LIN {X 0,Y 360.578,Z 690.318,A -85,B 0,C 180,E1 -13920.839,E2 -13920.839} C_VEL
LIN {X 0,Y 363.024,Z 692.376,A -85,B 0,C 180,E1 -13922.068,E2 -13922.068} C_VEL
LIN {X 0,Y 364.411,Z 693.279,A -85,B 0,C 180,E1 -13922.787,E2 -13922.787} C_VEL
LIN {X 0,Y 366.377,Z 696.293,A -85,B 0,C 180,E1 -13923.915,E2 -13923.915} C_VEL
LIN {X 0,Y 368.883,Z 698.376,A -85,B 0,C 180,E1 -13925.306,E2 -13925.306} C_VEL
LIN {X 0,Y 370.457,Z 699.391,A -85,B 0,C 180,E1 -13926.178,E2 -13926.178} C_VEL
LIN {X 0,Y 372.588,Z 702.531,A -85,B 0,C 180,E1 -13927.557,E2 -13927.557} C_VEL
LIN {X 0,Y 375.22,Z 704.628,A -85,B 0,C 180,E1 -13929.254,E2 -13929.254} C_VEL
LIN {X 0,Y 377.024,Z 705.757,A -85,B 0,C 180,E1 -13930.448,E2 -13930.448} C_VEL
LIN {X 0,Y 378.97,Z 708.665,A -85,B 0,C 180,E1 -13931.981,E2 -13931.981} C_VEL
LIN {X 0,Y 381.455,Z 710.749,A -85,B 0,C 180,E1 -13933.957,E2 -13933.957} C_VEL
LIN {X 0,Y 383.879,Z 712.198,A -85,B 0,C 180,E1 -13936.097,E2 -13936.097} C_VEL
LIN {X 0,Y 385.325,Z 714.601,A -85,B 0,C 180,E1 -13937.723,E2 -13937.723} C_VEL
LIN {X 0,Y 387.104,Z 716.368,A -85,B 0,C 180,E1 -13939.874,E2 -13939.874} C_VEL
LIN {X 0,Y 388.773,Z 717.316,A -85,B 0,C 180,E1 -13942.274,E2 -13942.274} C_VEL
LIN {X 0,Y 390.141,Z 718.042,A -85,B 0,C 180,E1 -13945.056,E2 -13945.056} C_VEL
LIN {X 0,Y 390.72,Z 718.32,A -85,B 0,C 180,E1 -13946.907,E2 -13946.907} C_VEL
LIN {X 0,Y 391.042,Z 718.625,A -85,B 0,C 180,E1 -13948.97,E2 -13948.97} C_VEL
LIN {X 0,Y 391.042,Z 718.628,A -85,B 0,C 180,E1 -13951.03,E2 -13951.03} C_VEL
LIN {X 0,Y 390.72,Z 718.32,A -85,B 0,C 180,E1 -13953.093,E2 -13953.093} C_VEL
LIN {X 0,Y 390.078,Z 717.948,A -85,B 0,C 180,E1 -13955.168,E2 -13955.168} C_VEL
LIN {X 0,Y 388.616,Z 717.21,A -85,B 0,C 180,E1 -13957.998,E2 -13957.998} C_VEL
LIN {X 0,Y 386.866,Z 716.144,A -85,B 0,C 180,E1 -13960.466,E2 -13960.466} C_VEL
LIN {X 0,Y 385.091,Z 714.233,A -85,B 0,C 180,E1 -13962.55,E2 -13962.55} C_VEL
LIN {X 0,Y 383.464,Z 711.736,A -85,B 0,C 180,E1 -13964.33,E2 -13964.33} C_VEL
LIN {X 0,Y 380.729,Z 710.261,A -85,B 0,C 180,E1 -13966.625,E2 -13966.625} C_VEL
LIN {X 0,Y 378.414,Z 707.927,A -85,B 0,C 180,E1 -13968.474,E2 -13968.474} C_VEL
LIN {X 0,Y 376.778,Z 705.402,A -85,B 0,C 180,E1 -13969.747,E2 -13969.747} C_VEL
LIN {X 0,Y 373.56,Z 703.487,A -85,B 0,C 180,E1 -13971.801,E2 -13971.801} C_VEL
LIN {X 0,Y 371.231,Z 700.802,A -85,B 0,C 180,E1 -13973.292,E2 -13973.292} C_VEL
LIN {X 0,Y 370.287,Z 699.091,A -85,B 0,C 180,E1 -13973.928,E2 -13973.928} C_VEL
LIN {X 0,Y 367.287,Z 697.223,A -85,B 0,C 180,E1 -13975.577,E2 -13975.577} C_VEL
LIN {X 0,Y 365.132,Z 694.577,A -85,B 0,C 180,E1 -13976.799,E2 -13976.799} C_VEL
LIN {X 0,Y 364.095,Z 692.896,A -85,B 0,C 180,E1 -13977.388,E2 -13977.388} C_VEL
LIN {X 0,Y 361.502,Z 691.284,A -85,B 0,C 180,E1 -13978.676,E2 -13978.676} C_VEL
LIN {X 0,Y 359.224,Z 688.533,A -85,B 0,C 180,E1 -13979.846,E2 -13979.846} C_VEL
LIN {X 0,Y 358.308,Z 686.907,A -85,B 0,C 180,E1 -13980.342,E2 -13980.342} C_VEL
LIN {X 0,Y 355.456,Z 685.116,A -85,B 0,C 180,E1 -13981.647,E2 -13981.647} C_VEL
LIN {X 0,Y 353.491,Z 682.584,A -85,B 0,C 180,E1 -13982.589,E2 -13982.589} C_VEL
LIN {X 0,Y 352.426,Z 680.85,A -85,B 0,C 180,E1 -13983.119,E2 -13983.119} C_VEL
LIN {X 0,Y 349.75,Z 679.112,A -85,B 0,C 180,E1 -13984.266,E2 -13984.266} C_VEL
LIN {X 0,Y 348.268,Z 676.877,A -85,B 0,C 180,E1 -13984.974,E2 -13984.974} C_VEL
LIN {X 0,Y 347.857,Z 675.498,A -85,B 0,C 180,E1 -13985.388,E2 -13985.388} C_VEL
LIN {X 0,Y 347.766,Z 674.995,A -85,B 0,C 180,E1 -13986.065,E2 -13986.065} C_VEL
LIN {X 0,Y 347.76,Z 674.98,A -85,B 0,C 180,E1 -13988.79,E2 -13988.79} C_VEL
LIN {X 0,Y 347.76,Z 674.981,A -85,B 0,C 180,E1 -13991.827,E2 -13991.827} C_VEL
LIN {X 0,Y 347.792,Z 674.977,A -85,B 0,C 180,E1 -13995.011,E2 -13995.011} C_VEL
LIN {X 0,Y 347.777,Z 674.978,A -85,B 0,C 180,E1 -13998.391,E2 -13998.391} C_VEL
LIN {X 0,Y 347.768,Z 674.952,A -85,B 0,C 180,E1 -14002.011,E2 -14002.011} C_VEL
LIN {X 0,Y 347.736,Z 674.953,A -85,B 0,C 180,E1 -14005.536,E2 -14005.536} C_VEL
LIN {X 0,Y 347.748,Z 674.942,A -85,B 0,C 180,E1 -14009.555,E2 -14009.555} C_VEL
LIN {X 0,Y 347.141,Z 675.009,A -85,B 0,C 180,E1 -14010.522,E2 -14010.522} C_VEL
LIN {X 0,Y 344.316,Z 675.368,A -85,B 0,C 180,E1 -14012.097,E2 -14012.097} C_VEL
LIN {X 0,Y 341.887,Z 675.687,A -85,B 0,C 180,E1 -14013.372,E2 -14013.372} C_VEL
LIN {X 0,Y 340.842,Z 675.832,A -85,B 0,C 180,E1 -14014.358,E2 -14014.358} C_VEL
LIN {X 0,Y 340.757,Z 675.844,A -85,B 0,C 180,E1 -14014.692,E2 -14014.692} C_VEL
LIN {X 0,Y 340.778,Z 675.835,A -85,B 0,C 180,E1 -14018.21,E2 -14018.21} C_VEL
LIN {X 0,Y 340.85,Z 675.822,A -85,B 0,C 180,E1 -14021.984,E2 -14021.984} C_VEL
LIN {X 0,Y 340.861,Z 675.829,A -85,B 0,C 180,E1 -14025.705,E2 -14025.705} C_VEL
LIN {X 0,Y 340.863,Z 675.834,A -85,B 0,C 180,E1 -14029.306,E2 -14029.306} C_VEL
LIN {X 0,Y 341.054,Z 675.797,A -85,B 0,C 180,E1 -14032.898,E2 -14032.898} C_VEL
LIN {X 0,Y 341.162,Z 675.779,A -85,B 0,C 180,E1 -14037.639,E2 -14037.639} C_VEL
LIN {X 0,Y 341.308,Z 675.782,A -85,B 0,C 180,E1 -14040,E2 -14040} C_VEL
LIN {X 0,Y 341.162,Z 675.783,A -85,B 0,C 180,E1 -14042.362,E2 -14042.362} C_VEL
LIN {X 0,Y 341.056,Z 675.795,A -85,B 0,C 180,E1 -14047.102,E2 -14047.102} C_VEL
LIN {X 0,Y 340.867,Z 675.836,A -85,B 0,C 180,E1 -14050.694,E2 -14050.694} C_VEL
LIN {X 0,Y 340.855,Z 675.831,A -85,B 0,C 180,E1 -14054.325,E2 -14054.325} C_VEL
LIN {X 0,Y 340.831,Z 675.827,A -85,B 0,C 180,E1 -14058.468,E2 -14058.468} C_VEL
LIN {X 0,Y 340.747,Z 675.838,A -85,B 0,C 180,E1 -14061.858,E2 -14061.858} C_VEL
LIN {X 0,Y 340.766,Z 675.842,A -85,B 0,C 180,E1 -14065.665,E2 -14065.665} C_VEL
LIN {X 0,Y 340.735,Z 675.794,A -85,B 0,C 180,E1 -14068.32,E2 -14068.32} C_VEL
LIN {X 0,Y 340.698,Z 675.83,A -85,B 0,C 180,E1 -14071.045,E2 -14071.045} C_VEL
LIN {X 0,Y 340.713,Z 675.82,A -85,B 0,C 180,E1 -14075.28,E2 -14075.28} C_VEL
LIN {X 0,Y 340.715,Z 675.857,A -85,B 0,C 180,E1 -14078.389,E2 -14078.389} C_VEL
LIN {X 0,Y 340.72,Z 675.826,A -85,B 0,C 180,E1 -14081.305,E2 -14081.305} C_VEL
LIN {X 0,Y 340.779,Z 676.004,A -85,B 0,C 180,E1 -14083.9,E2 -14083.9} C_VEL
LIN {X 0,Y 343.832,Z 686.497,A -85,B 0,C 180,E1 -14087.379,E2 -14087.379} C_VEL
LIN {X 0,Y 344.596,Z 688.812,A -85,B 0,C 180,E1 -14087.999,E2 -14087.999} C_VEL
LIN {X 0,Y 353.185,Z 704.061,A -85,B 0,C 180,E1 -14089.648,E2 -14089.648} C_VEL
LIN {X 0,Y 361.815,Z 720.686,A -85,B 0,C 180,E1 -14091.206,E2 -14091.206} C_VEL
LIN {X 0,Y 368.815,Z 735.619,A -85,B 0,C 180,E1 -14092.428,E2 -14092.428} C_VEL
LIN {X 0,Y 371.246,Z 747.626,A -85,B 0,C 180,E1 -14092.998,E2 -14092.998} C_VEL
LIN {X 0,Y 366.333,Z 892.343,A -85,B 0,C 180,E1 -14095.879,E2 -14095.879} C_VEL
LIN {X 0,Y 365.559,Z 904.031,A -85,B 0,C 180,E1 -14096.198,E2 -14096.198} C_VEL
LIN {X 0,Y 364.274,Z 917.366,A -85,B 0,C 180,E1 -14096.685,E2 -14096.685} C_VEL
LIN {X 0,Y 362.811,Z 930.484,A -85,B 0,C 180,E1 -14097.32,E2 -14097.32} C_VEL
LIN {X 0,Y 361.369,Z 941.872,A -85,B 0,C 180,E1 -14097.998,E2 -14097.998} C_VEL
LIN {X 0,Y 359.346,Z 955.107,A -85,B 0,C 180,E1 -14098.948,E2 -14098.948} C_VEL
LIN {X 0,Y 357.283,Z 967.494,A -85,B 0,C 180,E1 -14100.018,E2 -14100.018} C_VEL
LIN {X 0,Y 355.177,Z 978.841,A -85,B 0,C 180,E1 -14101.164,E2 -14101.164} C_VEL
LIN {X 0,Y 353.021,Z 989.641,A -85,B 0,C 180,E1 -14102.429,E2 -14102.429} C_VEL
LIN {X 0,Y 350.905,Z 1000.142,A -85,B 0,C 180,E1 -14103.857,E2 -14103.857} C_VEL
LIN {X 0,Y 348.96,Z 1009.413,A -85,B 0,C 180,E1 -14105.299,E2 -14105.299} C_VEL
LIN {X 0,Y 346.885,Z 1019.147,A -85,B 0,C 180,E1 -14107.045,E2 -14107.045} C_VEL
LIN {X 0,Y 345.045,Z 1027.671,A -85,B 0,C 180,E1 -14108.806,E2 -14108.806} C_VEL
LIN {X 0,Y 343.344,Z 1036.275,A -85,B 0,C 180,E1 -14110.883,E2 -14110.883} C_VEL
LIN {X 0,Y 342.102,Z 1042.707,A -85,B 0,C 180,E1 -14112.67,E2 -14112.67} C_VEL
LIN {X 0,Y 340.872,Z 1049.97,A -85,B 0,C 180,E1 -14115.066,E2 -14115.066} C_VEL
LIN {X 0,Y 340.227,Z 1054.624,A -85,B 0,C 180,E1 -14116.867,E2 -14116.867} C_VEL
LIN {X 0,Y 339.514,Z 1059.72,A -85,B 0,C 180,E1 -14119.263,E2 -14119.263} C_VEL
LIN {X 0,Y 339.209,Z 1063.72,A -85,B 0,C 180,E1 -14121.661,E2 -14121.661} C_VEL
LIN {X 0,Y 339.11,Z 1066.676,A -85,B 0,C 180,E1 -14124.052,E2 -14124.052} C_VEL
LIN {X 0,Y 339.028,Z 1067.86,A -85,B 0,C 180,E1 -14125.244,E2 -14125.244} C_VEL
LIN {X 0,Y 338.984,Z 1069.327,A -85,B 0,C 180,E1 -14127.624,E2 -14127.624} C_VEL
LIN {X 0,Y 339.064,Z 1069.815,A -85,B 0,C 180,E1 -14130,E2 -14130} C_VEL
LIN {X 0,Y 338.984,Z 1069.327,A -85,B 0,C 180,E1 -14132.376,E2 -14132.376} C_VEL
LIN {X 0,Y 339.028,Z 1067.86,A -85,B 0,C 180,E1 -14134.756,E2 -14134.756} C_VEL
LIN {X 0,Y 339.13,Z 1065.394,A -85,B 0,C 180,E1 -14137.143,E2 -14137.143} C_VEL
LIN {X 0,Y 339.419,Z 1060.808,A -85,B 0,C 180,E1 -14140.137,E2 -14140.137} C_VEL
LIN {X 0,Y 339.858,Z 1057.321,A -85,B 0,C 180,E1 -14141.934,E2 -14141.934} C_VEL
LIN {X 0,Y 340.529,Z 1052.312,A -85,B 0,C 180,E1 -14144.068,E2 -14144.068} C_VEL
LIN {X 0,Y 341.413,Z 1046.53,A -85,B 0,C 180,E1 -14146.134,E2 -14146.134} C_VEL
LIN {X 0,Y 342.98,Z 1038.5,A -85,B 0,C 180,E1 -14148.518,E2 -14148.518} C_VEL
LIN {X 0,Y 344.303,Z 1031.513,A -85,B 0,C 180,E1 -14150.304,E2 -14150.304} C_VEL
LIN {X 0,Y 345.932,Z 1023.543,A -85,B 0,C 180,E1 -14152.076,E2 -14152.076} C_VEL
LIN {X 0,Y 347.926,Z 1014.431,A -85,B 0,C 180,E1 -14153.827,E2 -14153.827} C_VEL
LIN {X 0,Y 350.037,Z 1004.176,A -85,B 0,C 180,E1 -14155.536,E2 -14155.536} C_VEL
LIN {X 0,Y 352.219,Z 993.996,A -85,B 0,C 180,E1 -14156.996,E2 -14156.996} C_VEL
LIN {X 0,Y 354.12,Z 983.826,A -85,B 0,C 180,E1 -14158.282,E2 -14158.282} C_VEL
LIN {X 0,Y 356.431,Z 972.159,A -85,B 0,C 180,E1 -14159.533,E2 -14159.533} C_VEL
LIN {X 0,Y 358.534,Z 960.134,A -85,B 0,C 180,E1 -14160.64,E2 -14160.64} C_VEL
LIN {X 0,Y 360.474,Z 947.814,A -85,B 0,C 180,E1 -14161.598,E2 -14161.598} C_VEL
LIN {X 0,Y 362.246,Z 935.271,A -85,B 0,C 180,E1 -14162.408,E2 -14162.408} C_VEL
LIN {X 0,Y 363.803,Z 921.842,A -85,B 0,C 180,E1 -14163.115,E2 -14163.115} C_VEL
LIN {X 0,Y 365.12,Z 908.926,A -85,B 0,C 180,E1 -14163.64,E2 -14163.64} C_VEL
LIN {X 0,Y 366.232,Z 894.922,A -85,B 0,C 180,E1 -14164.055,E2 -14164.055} C_VEL
LIN {X 0,Y 367.24,Z 866.824,A -85,B 0,C 180,E1 -14164.653,E2 -14164.653} C_VEL
LIN {X 0,Y 371.256,Z 746.985,A -85,B 0,C 180,E1 -14167.016,E2 -14167.016} C_VEL
LIN {X 0,Y 368.637,Z 735.279,A -85,B 0,C 180,E1 -14167.602,E2 -14167.602} C_VEL
LIN {X 0,Y 361.094,Z 719.093,A -85,B 0,C 180,E1 -14168.925,E2 -14168.925} C_VEL
LIN {X 0,Y 351.415,Z 700.875,A -85,B 0,C 180,E1 -14170.68,E2 -14170.68} C_VEL
LIN {X 0,Y 346.41,Z 692.124,A -85,B 0,C 180,E1 -14171.627,E2 -14171.627} C_VEL
LIN {X 0,Y 344.409,Z 688.353,A -85,B 0,C 180,E1 -14172.076,E2 -14172.076} C_VEL
LIN {X 0,Y 341.537,Z 678.501,A -85,B 0,C 180,E1 -14175.218,E2 -14175.218} C_VEL
LIN {X 0,Y 340.757,Z 675.869,A -85,B 0,C 180,E1 -14176.207,E2 -14176.207} C_VEL
LIN {X 0,Y 340.759,Z 675.826,A -85,B 0,C 180,E1 -14179.737,E2 -14179.737} C_VEL
LIN {X 0,Y 340.706,Z 675.822,A -85,B 0,C 180,E1 -14183.558,E2 -14183.558} C_VEL
LIN {X 0,Y 340.686,Z 675.846,A -85,B 0,C 180,E1 -14186.153,E2 -14186.153} C_VEL
LIN {X 0,Y 340.768,Z 675.793,A -85,B 0,C 180,E1 -14190.332,E2 -14190.332} C_VEL
LIN {X 0,Y 340.798,Z 675.805,A -85,B 0,C 180,E1 -14193.019,E2 -14193.019} C_VEL
LIN {X 0,Y 340.749,Z 675.853,A -85,B 0,C 180,E1 -14195.638,E2 -14195.638} C_VEL
LIN {X 0,Y 340.758,Z 675.851,A -85,B 0,C 180,E1 -14199.475,E2 -14199.475} C_VEL
LIN {X 0,Y 340.851,Z 675.823,A -85,B 0,C 180,E1 -14201.984,E2 -14201.984} C_VEL
LIN {X 0,Y 340.862,Z 675.832,A -85,B 0,C 180,E1 -14205.704,E2 -14205.704} C_VEL
LIN {X 0,Y 340.867,Z 675.837,A -85,B 0,C 180,E1 -14209.306,E2 -14209.306} C_VEL
LIN {X 0,Y 341.056,Z 675.795,A -85,B 0,C 180,E1 -14212.898,E2 -14212.898} C_VEL
LIN {X 0,Y 341.162,Z 675.782,A -85,B 0,C 180,E1 -14217.638,E2 -14217.638} C_VEL
LIN {X 0,Y 341.308,Z 675.781,A -85,B 0,C 180,E1 -14220,E2 -14220} C_VEL
LIN {X 0,Y 341.162,Z 675.778,A -85,B 0,C 180,E1 -14222.361,E2 -14222.361} C_VEL
LIN {X 0,Y 341.054,Z 675.799,A -85,B 0,C 180,E1 -14227.102,E2 -14227.102} C_VEL
LIN {X 0,Y 340.863,Z 675.836,A -85,B 0,C 180,E1 -14230.694,E2 -14230.694} C_VEL
LIN {X 0,Y 340.854,Z 675.831,A -85,B 0,C 180,E1 -14234.325,E2 -14234.325} C_VEL
LIN {X 0,Y 340.83,Z 675.828,A -85,B 0,C 180,E1 -14238.467,E2 -14238.467} C_VEL
LIN {X 0,Y 340.748,Z 675.839,A -85,B 0,C 180,E1 -14241.858,E2 -14241.858} C_VEL
